(* Logix 5000 project; controller LeakTestAuto vendor 1 type 14 code 226 rev 37.11; software revision 37.01; part 13 of 15 *)
(* tags used below, declared in another part *)
   AOI_CapShuffle_Seq : AOI_Sequencer_x64;
   AOI_CTS1 : AOI_CTS_INSTRUMENT;
   AOI_CTS2 : AOI_CTS_INSTRUMENT;
   AOI_RobotPos : AOI_RobotPositions;
   AOI_SeqSteps : AOI_StandardSeqSteps;
   BarcodeInputs : udt_KeyenceScannerInputs;
   BarcodeScanner : udt_OutputStructure;
   CapShuffle_CTS1Bad : COUNTER;
   CapShuffle_CTS1Good : COUNTER;
   CapShuffle_CTS2Bad : COUNTER;
   CapShuffle_CTS2Good : COUNTER;
   CapShuffle_Seq : udt_SequenceStructure_X64;
   Conveyor : udt_OutputStructure;
   Conveyor_Seq : udt_SequenceStructure_X64;
   ConveyorHomeCounter : COUNTER;
   CTS1_Seq : udt_SequenceStructure_X64;
   CTS2_Seq : udt_SequenceStructure_X64;
   FaultsAndWarnings : STRING[96];
   LeakTester1 : udt_OutputStructure;
   LeakTester2 : udt_OutputStructure;
   Nest1Cylinder : udt_OutputStructure;
   Nest1Empty : BOOL;
   Nest1Ready : BOOL;
   Nest2Cylinder : udt_OutputStructure;
   Nest2Empty : BOOL;
   Nest2Ready : BOOL;
   OP220 : udt_Mode;
   OP220_HomingSeq : udt_SequenceStructure_X64;
   OP220_Seq : udt_SequenceStructure_X64;
   Robot : udt_OutputStructure;
   RobotGripper : udt_OutputStructure;
   RobotInputs : udt_EpsonInputs;
   ShiftTimes : SINT[24];
   TempStrBuff : STRING[10];
   test : BOOL;
   TON_CapShuffleCTS1Delay : TIMER;
   TON_CapShuffleCTS2Delay : TIMER;
   AOI_IOCounter : AOI_IOCounter;
   I_OP220_N3_CONVEYOR_CLEAT : ALIAS FOR Local:3:I.Pt13.Data;
   I_OP220_N3_CONVEYOR_LOAD : ALIAS FOR Local:3:I.Pt12.Data;
   I_OP220_N3_CONVEYOR_UNLOAD : ALIAS FOR Local:3:I.Pt14.Data;
   I_OP220_N3_DUT_PRE_NEST_0 : ALIAS FOR Local:3:I.Pt00.Data;
   I_OP220_N3_DUT_PRE_NEST_1 : ALIAS FOR Local:3:I.Pt01.Data;
   I_OP220_N3_DUT_PRE_NEST_2 : ALIAS FOR Local:3:I.Pt02.Data;
   I_OP220_N3_MAIN_AIR_OK : ALIAS FOR Local:3:I.Pt07.Data;
   I_OP220_N3_NEST1_EXTEND : ALIAS FOR Local:3:I.Pt04.Data;
   I_OP220_N3_NEST1_HOME : ALIAS FOR Local:3:I.Pt03.Data;
   I_OP220_N3_NEST2_EXTEND : ALIAS FOR Local:3:I.Pt06.Data;
   I_OP220_N3_NEST2_HOME : ALIAS FOR Local:3:I.Pt05.Data;
   I_OP220_N3_REJECT_BIN_OK : ALIAS FOR Local:3:I.Pt09.Data;
   I_OP220_N3_REJECT_CHUTE_PART : ALIAS FOR Local:3:I.Pt10.Data;
   I_OP220_N4_AC_SURGE_OK : ALIAS FOR Local:4:I.Pt00.Data;
   I_OP220_N4_CONVEYOR_ALARM_OK : ALIAS FOR Local:4:I.Pt03.Data;
   I_OP220_N4_CONVEYOR_SPEED : ALIAS FOR Local:4:I.Pt02.Data;
   I_OP220_N4_DC_OK : ALIAS FOR Local:4:I.Pt01.Data;
   I_OP220_N4_DC_OK_PS2 : ALIAS FOR Local:4:I.Pt04.Data;
   IOCounterHasRef : BOOL;
   IOCounterLastData : INT[8];
   IOLabels : STRING[128];
   IOResetArray : INT[8];
   IOTriggerCounts : UDINT[128];
   NoData : AB:5000_DI16:I:0;
   O_OP220_N5_CONV_FWD : ALIAS FOR Local:5:O.Pt12.Data;
   O_OP220_N5_CONV_REV : ALIAS FOR Local:5:O.Pt11.Data;
   O_OP220_N5_EN_CONV_ALM_RST : ALIAS FOR Local:5:O.Pt10.Data;
   O_OP220_N5_EN_GRIPPER_GRIP : ALIAS FOR Local:5:O.Pt14.Data;
   O_OP220_N5_EN_GRIPPER_UNGRIP : ALIAS FOR Local:5:O.Pt15.Data;
   O_OP220_N5_EN_LT_BU : ALIAS FOR Local:5:O.Pt03.Data;
   O_OP220_N5_EN_LT_GN : ALIAS FOR Local:5:O.Pt00.Data;
   O_OP220_N5_EN_LT_RD : ALIAS FOR Local:5:O.Pt02.Data;
   O_OP220_N5_EN_LT_YE : ALIAS FOR Local:5:O.Pt01.Data;
   O_OP220_N5_EN_MAIN_AIR : ALIAS FOR Local:5:O.Pt04.Data;
   O_OP220_N5_EN_NEST1_EXT : ALIAS FOR Local:5:O.Pt05.Data;
   O_OP220_N5_EN_NEST1_HOME : ALIAS FOR Local:5:O.Pt06.Data;
   O_OP220_N5_EN_NEST2_EXT : ALIAS FOR Local:5:O.Pt07.Data;
   O_OP220_N5_EN_NEST2_HOME : ALIAS FOR Local:5:O.Pt08.Data;
   O_OP220_N5_EN_ROBOT_LATCHOFF : ALIAS FOR Local:5:O.Pt09.Data;
   PLC : AOI_PLC;
   SI_OP220_N1_CTRL_VLAVE_NC1 : ALIAS FOR Local:1:I.Pt04.Data;
   SI_OP220_N1_LASER_AREA_NC12 : ALIAS FOR Local:1:I.Pt00.Data;
   SI_OP220_N1_LASER_GUARD_NC12 : ALIAS FOR Local:1:I.Pt01.Data;
   SI_OP220_N1_SSR_12 : ALIAS FOR Local:1:I.Pt03.Data;
   SO_OP220_N2_SSR_1 : ALIAS FOR Local:2:O.Pt00.Data;
   SO_OP220_N2_SSR_2 : ALIAS FOR Local:2:O.Pt01.Data;
(* MainProgram, continued *)

ROUTINE R98_IOCounter   (* ladder *)
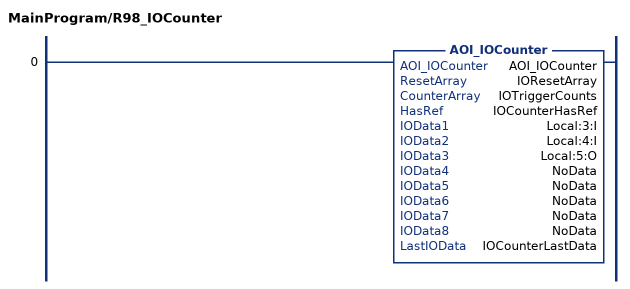
   0: AOI_IOCounter(AOI_IOCounter,IOResetArray,IOTriggerCounts,IOCounterHasRef,Local:3:I,Local:4:I,Local:5:O,NoData,NoData,NoData,NoData,NoData,IOCounterLastData);
END_ROUTINE

ROUTINE R999_SetConstants   (* structured text *)
   if PLC.FirstScan then
   	// [1] IB8S
   	IOLabels[000] := 'SI_OP220_N1_LASER_AREA_NC12';
   	IOLabels[001] := 'SI_OP220_N1_LASER_GUARD_NC12';
   	IOLabels[002] := '';
   	IOLabels[003] := 'SI_OP220_N1_SSR_12';
   	IOLabels[004] := 'SI_OP220_N1_CTRL_VLAVE_NC1';
   	IOLabels[005] := '';
   	IOLabels[006] := '';
   	IOLabels[007] := '';
   	// [2] OBV8S
   	IOLabels[008] := 'SO_OP220_N2_SSR_1';
   	IOLabels[009] := 'SO_OP220_N2_SSR_2';
   	IOLabels[010] := '';
   	IOLabels[011] := '';
   	IOLabels[012] := '';
   	IOLabels[013] := '';
   	IOLabels[014] := '';
   	IOLabels[015] := '';
   	// [3] IB16
   	IOLabels[016] := 'I_OP220_N3_DUT_PRE_NEST_0';
   	IOLabels[017] := 'I_OP220_N3_DUT_PRE_NEST_1';
   	IOLabels[018] := 'I_OP220_N3_DUT_PRE_NEST_2';
   	IOLabels[019] := 'I_OP220_N3_NEST1_HOME';
   	IOLabels[020] := 'I_OP220_N3_NEST1_EXTEND';
   	IOLabels[021] := 'I_OP220_N3_NEST2_HOME';
   	IOLabels[022] := 'I_OP220_N3_NEST2_EXTEND';
   	IOLabels[023] := 'I_OP220_N3_MAIN_AIR_OK';
   	IOLabels[024] := '';
   	IOLabels[025] := 'I_OP220_N3_REJECT_BIN_OK';
   	IOLabels[026] := 'I_OP220_N3_REJECT_CHUTE_PART';
   	IOLabels[027] := '';
   	IOLabels[028] := 'I_OP220_N3_CONVEYOR_LOAD';
   	IOLabels[029] := 'I_OP220_N3_CONVEYOR_CLEAT';
   	IOLabels[030] := 'I_OP220_N3_CONVEYOR_UNLOAD';
   	IOLabels[031] := '';
   	// [4] IB16
   	IOLabels[032] := 'I_OP220_N4_AC_SURGE_OK';
   	IOLabels[033] := 'I_OP220_N4_DC_OK';
   	IOLabels[034] := 'I_OP220_N4_CONVEYOR_SPEED';
   	IOLabels[035] := 'I_OP220_N4_CONVEYOR_ALARM_OK';
   	IOLabels[036] := 'I_OP220_N4_DC_OK_PS2';
   	IOLabels[037] := '';
   	IOLabels[038] := '';
   	IOLabels[039] := '';
   	IOLabels[040] := '';
   	IOLabels[041] := '';
   	IOLabels[042] := '';
   	IOLabels[043] := '';
   	IOLabels[044] := '';
   	IOLabels[045] := '';
   	IOLabels[046] := '';
   	IOLabels[047] := '';
   	// [5] OB16
   	IOLabels[048] := 'O_OP220_N5_EN_LT_GN';
   	IOLabels[049] := 'O_OP220_N5_EN_LT_YE';
   	IOLabels[050] := 'O_OP220_N5_EN_LT_RD';
   	IOLabels[051] := 'O_OP220_N5_EN_LT_BU';
   	IOLabels[052] := 'O_OP220_N5_EN_MAIN_AIR';
   	IOLabels[053] := 'O_OP220_N5_EN_NEST1_EXT';
   	IOLabels[054] := 'O_OP220_N5_EN_NEST1_HOME';
   	IOLabels[055] := 'O_OP220_N5_EN_NEST2_EXT';
   	IOLabels[056] := 'O_OP220_N5_EN_NEST2_HOME';
   	IOLabels[057] := 'O_OP220_N5_EN_ROBOT_LATCHOFF';
   	IOLabels[058] := 'O_OP220_N5_EN_CONV_ALM_RST';
   	IOLabels[059] := 'O_OP220_N5_CONV_REV';
   	IOLabels[060] := 'O_OP220_N5_CONV_FWD';
   	IOLabels[061] := '';
   	IOLabels[062] := 'O_OP220_N5_EN_GRIPPER_GRIP';
   	IOLabels[063] := 'O_OP220_N5_EN_GRIPPER_UNGRIP';
   	IOLabels[064] := '';
   	IOLabels[065] := '';
   	IOLabels[066] := '';
   	IOLabels[067] := '';
   	IOLabels[068] := '';
   	IOLabels[069] := '';
   	IOLabels[070] := '';
   	IOLabels[071] := '';
   	IOLabels[072] := '';
   	IOLabels[073] := '';
   	IOLabels[074] := '';
   	IOLabels[075] := '';
   	IOLabels[076] := '';
   	IOLabels[077] := '';
   	IOLabels[078] := '';
   	IOLabels[079] := '';
   	IOLabels[080] := '';
   	IOLabels[081] := '';
   	IOLabels[082] := '';
   	IOLabels[083] := '';
   	IOLabels[084] := '';
   	IOLabels[085] := '';
   	IOLabels[086] := '';
   	IOLabels[087] := '';
   	IOLabels[088] := '';
   	IOLabels[089] := '';
   	IOLabels[090] := '';
   	IOLabels[091] := '';
   	IOLabels[092] := '';
   	IOLabels[093] := '';
   	IOLabels[094] := '';
   	IOLabels[095] := '';
   	IOLabels[096] := '';
   	IOLabels[097] := '';
   	IOLabels[098] := '';
   	IOLabels[099] := '';
   	IOLabels[100] := '';
   	IOLabels[101] := '';
   	IOLabels[102] := '';
   	IOLabels[103] := '';
   	IOLabels[104] := '';
   	IOLabels[105] := '';
   	IOLabels[106] := '';
   	IOLabels[107] := '';
   	IOLabels[108] := '';
   	IOLabels[109] := '';
   	IOLabels[110] := '';
   	IOLabels[111] := '';
   	IOLabels[112] := '';
   	IOLabels[113] := '';
   	IOLabels[114] := '';
   	IOLabels[115] := '';
   	IOLabels[116] := '';
   	IOLabels[117] := '';
   	IOLabels[118] := '';
   	IOLabels[119] := '';
   	IOLabels[120] := '';
   	IOLabels[121] := '';
   	IOLabels[122] := '';
   	IOLabels[123] := '';
   	IOLabels[124] := '';
   	IOLabels[125] := '';
   	IOLabels[126] := '';
   	IOLabels[127] := '';
   
   	ShiftTimes[0] := 7;
   	ShiftTimes[1] := 15;
   	ShiftTimes[2] := 23;
   	ShiftTimes[3] := -1;
   	ShiftTimes[4] := -1;
   	ShiftTimes[5] := -1;
   	ShiftTimes[6] := -1;
   	ShiftTimes[7] := -1;
   	ShiftTimes[8] := -1;
   	ShiftTimes[9] := -1;
   	ShiftTimes[10] := -1;
   	ShiftTimes[11] := -1;
   	ShiftTimes[12] := -1;
   	ShiftTimes[13] := -1;
   	ShiftTimes[14] := -1;
   	ShiftTimes[15] := -1;
   	ShiftTimes[16] := -1;
   	ShiftTimes[17] := -1;
   	ShiftTimes[18] := -1;
   	ShiftTimes[19] := -1;
   	ShiftTimes[20] := -1;
   	ShiftTimes[21] := -1;
   	ShiftTimes[22] := -1;
   	ShiftTimes[23] := -1;
   
   	// System Faults
   	FaultsAndWarnings[000] := 'Main power off';
   	FaultsAndWarnings[001] := 'Main air not OK';
   	FaultsAndWarnings[002] := 'EStop high';
   	FaultsAndWarnings[003] := 'Guard doors open';
   	FaultsAndWarnings[004] := 'Reject bin missing';
   	FaultsAndWarnings[005] := 'No EIP connection to barcode scanner';
   	FaultsAndWarnings[006] := 'No EIP connection to CTS1';
   	FaultsAndWarnings[007] := 'No EIP connection to CTS2';
   	FaultsAndWarnings[008] := 'No EIP connection to Robot';
   	FaultsAndWarnings[009] := 'EStop Safety Block faulted';
   	FaultsAndWarnings[010] := 'Barcode scanner fault';
   	FaultsAndWarnings[011] := 'CTS1 fault';
   	FaultsAndWarnings[012] := 'CTS2 fault';
   	FaultsAndWarnings[013] := 'Robot fault';
   	FaultsAndWarnings[014] := 'Robot gripper in unknown state';
   	FaultsAndWarnings[015] := 'Conveyor alarm high';
   	FaultsAndWarnings[016] := 'Cylinder 1 fault';
   	FaultsAndWarnings[017] := 'Cylinder 2 fault';
   	FaultsAndWarnings[018] := '24V DC not OK';
   	FaultsAndWarnings[019] := 'Check conveyor cleat sensor';
   	FaultsAndWarnings[020] := '';
   	FaultsAndWarnings[021] := '';
   	FaultsAndWarnings[022] := '';
   	FaultsAndWarnings[023] := '';
   	FaultsAndWarnings[024] := '';
   	FaultsAndWarnings[025] := '';
   	FaultsAndWarnings[026] := '';
   	FaultsAndWarnings[027] := '';
   	FaultsAndWarnings[028] := '';
   	FaultsAndWarnings[029] := '';
   	FaultsAndWarnings[030] := '';
   	FaultsAndWarnings[031] := '';
   	// Sequence Faults
   	FaultsAndWarnings[032] := '3 in a row fault';
   	FaultsAndWarnings[033] := '5 in an hour fault';
   	FaultsAndWarnings[034] := '10 in a shift fault';
   	FaultsAndWarnings[035] := '';
   	FaultsAndWarnings[036] := '';
   	FaultsAndWarnings[037] := '';
   	FaultsAndWarnings[038] := '';
   	FaultsAndWarnings[039] := '';
   	FaultsAndWarnings[040] := '';
   	FaultsAndWarnings[041] := '';
   	FaultsAndWarnings[042] := 'Homing cycle overtime';
   	FaultsAndWarnings[043] := 'Fail chute failed to register unit (Homing Seq)';
   	FaultsAndWarnings[044] := 'Fail chute failed to register unit (Auto Seq)';
   	FaultsAndWarnings[045] := 'Cylinder 1 down timeout';
   	FaultsAndWarnings[046] := 'Cylinder 2 down timeout';
   	FaultsAndWarnings[047] := 'Cylinder 1 up timeout';
   	FaultsAndWarnings[048] := 'Cylinder 2 up timeout';
   	FaultsAndWarnings[049] := 'Cylinder 1 movement requested but RFID not matching expected value.';
   	FaultsAndWarnings[050] := 'Cylinder 2 movement requested but RFID not matching expected value.';
   	FaultsAndWarnings[051] := '';
   	FaultsAndWarnings[052] := '';
   	FaultsAndWarnings[053] := '';
   	FaultsAndWarnings[054] := '';
   	FaultsAndWarnings[055] := '';
   	FaultsAndWarnings[056] := '';
   	FaultsAndWarnings[057] := '';
   	FaultsAndWarnings[058] := '';
   	FaultsAndWarnings[059] := '';
   	FaultsAndWarnings[060] := '';
   	FaultsAndWarnings[061] := '';
   	FaultsAndWarnings[062] := '';
   	FaultsAndWarnings[063] := '';
   	// Warnings
   	FaultsAndWarnings[064] := 'Cycle stop requested';
   	FaultsAndWarnings[065] := 'Cycle pause requested';
   	FaultsAndWarnings[066] := 'Step mode active';
   	FaultsAndWarnings[067] := 'Dry cycle active';
   	FaultsAndWarnings[068] := 'MES bypass active';
   	FaultsAndWarnings[069] := '';
   	FaultsAndWarnings[070] := '';
   	FaultsAndWarnings[071] := '';
   	FaultsAndWarnings[072] := '';
   	FaultsAndWarnings[073] := '';
   	FaultsAndWarnings[074] := 'Main sequence stuck on step$n';
   	FaultsAndWarnings[075] := 'Homing sequence stuck on step$n';
   	FaultsAndWarnings[076] := 'CTS1 sequence stuck on step ';
   	FaultsAndWarnings[077] := 'CTS2 sequence stuck on step ';
   	FaultsAndWarnings[078] := 'Conveyor sequence stuck on step ';
   	FaultsAndWarnings[079] := 'Main sequence stuck on step$n';
   	FaultsAndWarnings[080] := 'Homing sequence stuck on step$n';
   	FaultsAndWarnings[081] := 'CTS1 sequence stuck on step ';
   	FaultsAndWarnings[082] := 'CTS2 sequence stuck on step ';
   	FaultsAndWarnings[083] := 'Conveyor sequence stuck on step ';
   	FaultsAndWarnings[084] := 'CTS1 test requested but interlock not met';
   	FaultsAndWarnings[085] := 'CTS2 test requested but interlock not met';
   	FaultsAndWarnings[086] := 'CTS1 not ready';
   	FaultsAndWarnings[087] := 'CTS2 not ready';
   	FaultsAndWarnings[088] := 'Robot movement requested but interlock not met';
   	FaultsAndWarnings[089] := 'Conveyor movement requested but interlock not met';
   	FaultsAndWarnings[090] := 'Nest 1 movement requested but interlock not met';
   	FaultsAndWarnings[091] := 'Nest 2 movement requested but interlock not met';
   	FaultsAndWarnings[092] := '';
   	FaultsAndWarnings[093] := '';
   	FaultsAndWarnings[094] := 'Fail bin full, please empty';
   	FaultsAndWarnings[095] := '';
   end_if;
   
   // Done this way because concat cannot accept string literals
   // DTOS(OP220_Seq.CurrentStep,TempStrBuff[0]);
   // CONCAT(FaultsAndWarnings[079], TempStrBuff[0], FaultsAndWarnings[074]);
   CONCAT(FaultsAndWarnings[079], OP220_Seq.HMI_CurrentStepDescription, FaultsAndWarnings[074]);
   // DTOS(OP220_HomingSeq.CurrentStep,TempStrBuff[0]);
   // CONCAT(FaultsAndWarnings[080], TempStrBuff[0], FaultsAndWarnings[075]);
   CONCAT(FaultsAndWarnings[080], OP220_HomingSeq.HMI_CurrentStepDescription, FaultsAndWarnings[075]);
   DTOS(CTS1_Seq.CurrentStep,TempStrBuff[0]);
   CONCAT(FaultsAndWarnings[081], TempStrBuff[0], FaultsAndWarnings[076]);
   DTOS(CTS2_Seq.CurrentStep,TempStrBuff[0]);
   CONCAT(FaultsAndWarnings[082], TempStrBuff[0], FaultsAndWarnings[077]);
   DTOS(Conveyor_Seq.CurrentStep,TempStrBuff[0]);
   CONCAT(FaultsAndWarnings[083], TempStrBuff[0], FaultsAndWarnings[078]);
   
   AOI_RobotPositions(AOI_RobotPos);
   AOI_StandardSeqSteps(AOI_SeqSteps);
END_ROUTINE

ROUTINE R99_StepDescriptions   (* structured text *)
   case OP220_Seq.CurrentStep of
   	1000:
   		OP220_Seq.HMI_CurrentStepDescription := 'Waiting for next action';
   	2000,2010,2500,2510:
   		OP220_Seq.HMI_CurrentStepDescription := 'Pick up DUT from load nest';
   	2020,2030,2520,2530:
   		OP220_Seq.HMI_CurrentStepDescription := 'Scan DUT barcode';
   	2040,2050,2060:
   		OP220_Seq.HMI_CurrentStepDescription := 'Load DUT to nest 1';
   	2540,2550,2560:
   		OP220_Seq.HMI_CurrentStepDescription := 'Load DUT to nest 2';
   	2070,2080:
   		OP220_Seq.HMI_CurrentStepDescription := 'Start leak test nest 1';
   	2570,2580:
   		OP220_Seq.HMI_CurrentStepDescription := 'Start leak test nest 2';
   	3000,3010:
   		OP220_Seq.HMI_CurrentStepDescription := 'Pick up DUT from nest 1';
   	3500,3510:
   		OP220_Seq.HMI_CurrentStepDescription := 'Pick up DUT from nest 2';
   	3020,3520:
   		OP220_Seq.HMI_CurrentStepDescription := 'Drop off DUT';
   	3030,3040,3530,3540:
   		OP220_Seq.HMI_CurrentStepDescription := 'Drop off DUT at conveyor';
   	3050,3550:
   		OP220_Seq.HMI_CurrentStepDescription := 'Index conveyor';
   	7000,7010:
   		OP220_Seq.HMI_CurrentStepDescription := 'Drop off DUT at fail chute (Barcode)';
   	7100,7110:
   		OP220_Seq.HMI_CurrentStepDescription := 'Drop off DUT at fail chute (Nest 1)';
   	7200,7210:
   		OP220_Seq.HMI_CurrentStepDescription := 'Drop off DUT at fail chute (Nest 2)';
   	else
   		OP220_Seq.HMI_CurrentStepDescription := '';
   end_case;
   
   case OP220_HomingSeq.CurrentStep of
   	1000,1010:
   		OP220_HomingSeq.HMI_CurrentStepDescription := 'Drop gripped DUT to fail chute';
   	1020,1030:
   		OP220_HomingSeq.HMI_CurrentStepDescription := 'Move nest cylinders to home position';
   	1040,1050,1060,1070:
   		OP220_HomingSeq.HMI_CurrentStepDescription := 'Unload nest 1 to fail chute';
   	1080,1090,1100,1110:
   		OP220_HomingSeq.HMI_CurrentStepDescription := 'Unload nest 2 to fail chute';
   	1120,1130:
   		OP220_HomingSeq.HMI_CurrentStepDescription := 'Move robot to scanner';
   	1140,1150:
   		OP220_HomingSeq.HMI_CurrentStepDescription := 'Check conveyor empty (';
   		DTOS(ConveyorHomeCounter.ACC, TempStrBuff[0]);
   		TempStrBuff[1] := '/';
   		DTOS(ConveyorHomeCounter.PRE, TempStrBuff[2]);
   		TempStrBuff[3] := ')';
   		CONCAT(OP220_HomingSeq.HMI_CurrentStepDescription, TempStrBuff[0], OP220_HomingSeq.HMI_CurrentStepDescription);
   		CONCAT(OP220_HomingSeq.HMI_CurrentStepDescription, TempStrBuff[1], OP220_HomingSeq.HMI_CurrentStepDescription);
   		CONCAT(OP220_HomingSeq.HMI_CurrentStepDescription, TempStrBuff[2], OP220_HomingSeq.HMI_CurrentStepDescription);
   		CONCAT(OP220_HomingSeq.HMI_CurrentStepDescription, TempStrBuff[3], OP220_HomingSeq.HMI_CurrentStepDescription);
   	else
   		OP220_HomingSeq.HMI_CurrentStepDescription := '';
   end_case;
END_ROUTINE

ROUTINE zR10_CapShuffle   (* ladder *)
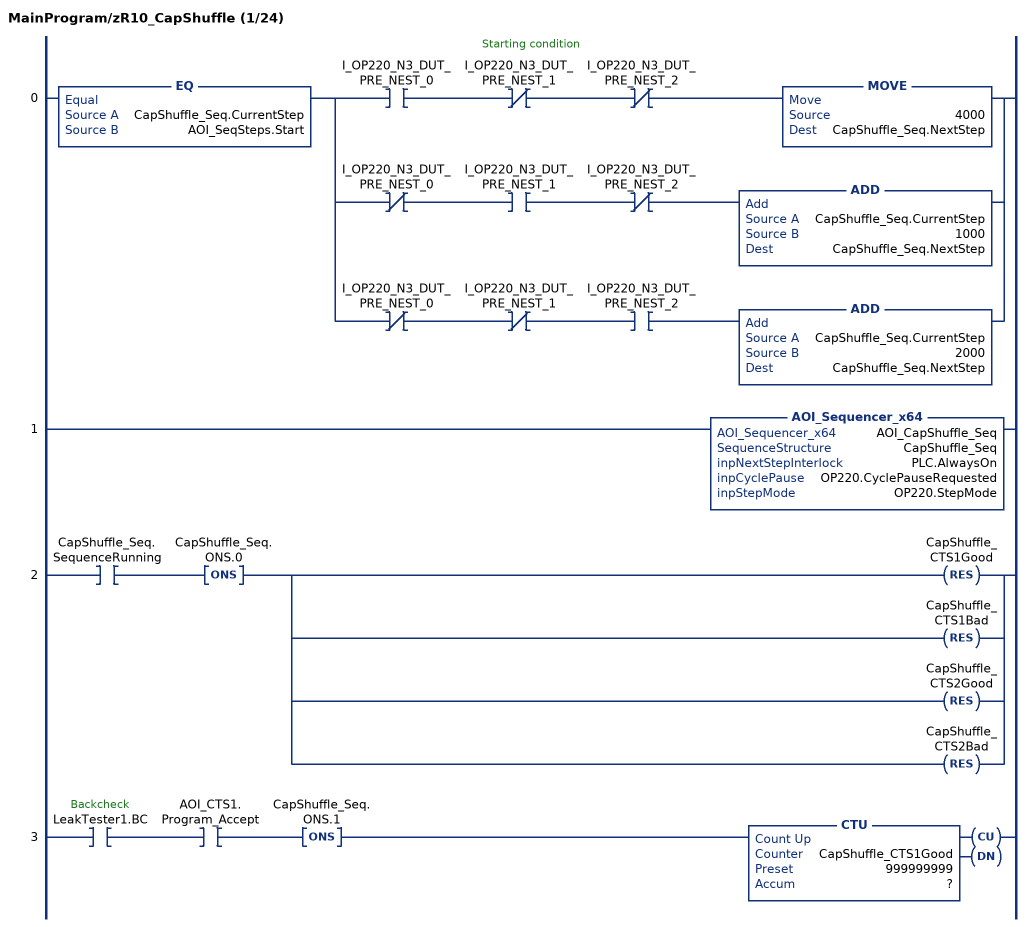
   // Starting condition
   0: EQ(CapShuffle_Seq.CurrentStep,AOI_SeqSteps.Start)[XIC(I_OP220_N3_DUT_PRE_NEST_0) XIO(I_OP220_N3_DUT_PRE_NEST_1) XIO(I_OP220_N3_DUT_PRE_NEST_2) MOVE(4000,CapShuffle_Seq.NextStep) ,XIO(I_OP220_N3_DUT_PRE_NEST_0) XIC(I_OP220_N3_DUT_PRE_NEST_1) XIO(I_OP220_N3_DUT_PRE_NEST_2) ADD(CapShuffle_Seq.CurrentStep,1000,CapShuffle_Seq.NextStep) ,XIO(I_OP220_N3_DUT_PRE_NEST_0) XIO(I_OP220_N3_DUT_PRE_NEST_1) XIC(I_OP220_N3_DUT_PRE_NEST_2) ADD(CapShuffle_Seq.CurrentStep,2000,CapShuffle_Seq.NextStep) ];
   1: AOI_Sequencer_x64(AOI_CapShuffle_Seq,CapShuffle_Seq,PLC.AlwaysOn,OP220.CyclePauseRequested,OP220.StepMode);
   2: XIC(CapShuffle_Seq.SequenceRunning)ONS(CapShuffle_Seq.ONS.0)[RES(CapShuffle_CTS1Good) ,RES(CapShuffle_CTS1Bad) ,RES(CapShuffle_CTS2Good) ,RES(CapShuffle_CTS2Bad) ];
   3: XIC(LeakTester1.BC)XIC(AOI_CTS1.Program_Accept)ONS(CapShuffle_Seq.ONS.1)CTU(CapShuffle_CTS1Good,?,?);
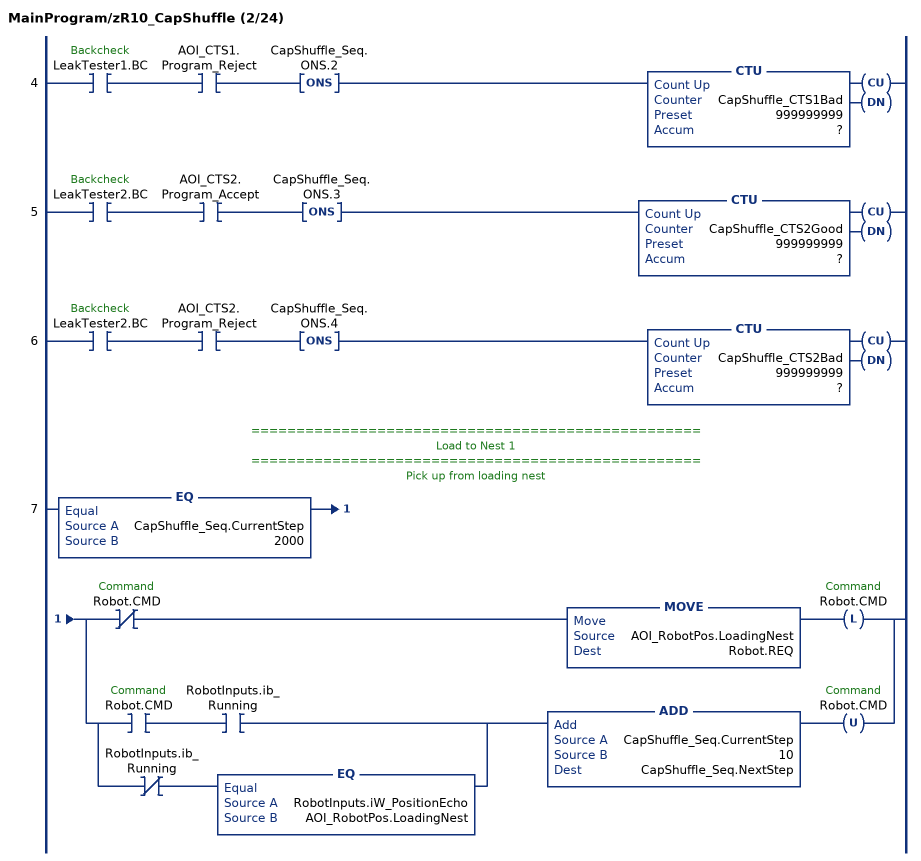
   4: XIC(LeakTester1.BC)XIC(AOI_CTS1.Program_Reject)ONS(CapShuffle_Seq.ONS.2)CTU(CapShuffle_CTS1Bad,?,?);
   5: XIC(LeakTester2.BC)XIC(AOI_CTS2.Program_Accept)ONS(CapShuffle_Seq.ONS.3)CTU(CapShuffle_CTS2Good,?,?);
   6: XIC(LeakTester2.BC)XIC(AOI_CTS2.Program_Reject)ONS(CapShuffle_Seq.ONS.4)CTU(CapShuffle_CTS2Bad,?,?);
   // ==================================================
   // Load to Nest 1
   // ==================================================
   // Pick up from loading nest
   7: EQ(CapShuffle_Seq.CurrentStep,2000)[XIO(Robot.CMD) MOVE(AOI_RobotPos.LoadingNest,Robot.REQ) OTL(Robot.CMD) ,[XIC(Robot.CMD) XIC(RobotInputs.ib_Running) ,XIO(RobotInputs.ib_Running) EQ(RobotInputs.iW_PositionEcho,AOI_RobotPos.LoadingNest) ] ADD(CapShuffle_Seq.CurrentStep,10,CapShuffle_Seq.NextStep) OTU(Robot.CMD) ];
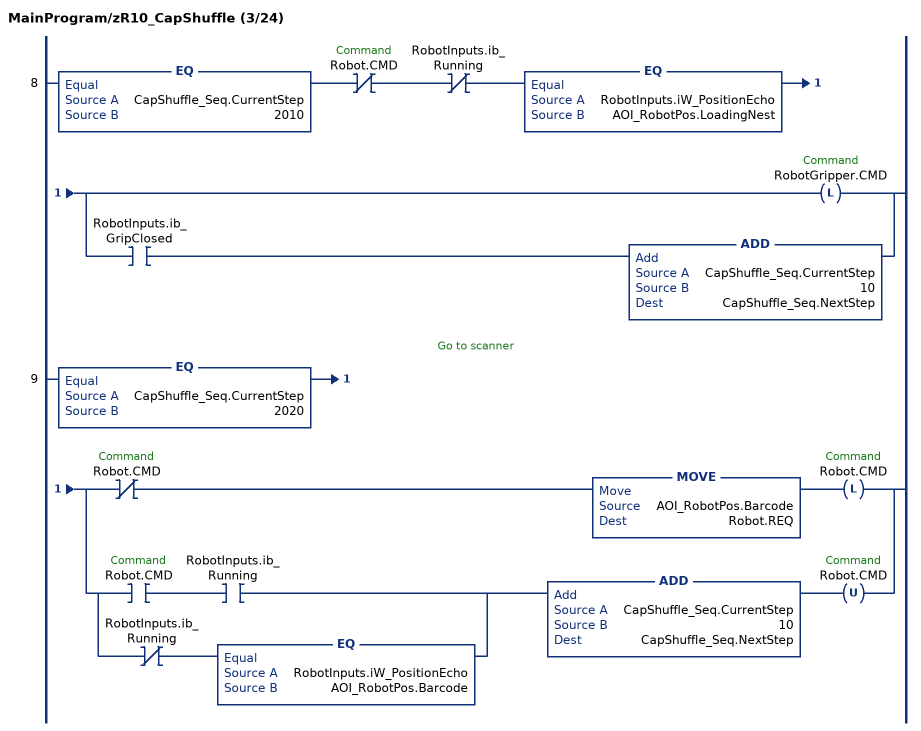
   8: EQ(CapShuffle_Seq.CurrentStep,2010)XIO(Robot.CMD)XIO(RobotInputs.ib_Running)EQ(RobotInputs.iW_PositionEcho,AOI_RobotPos.LoadingNest)[OTL(RobotGripper.CMD) ,XIC(RobotInputs.ib_GripClosed) ADD(CapShuffle_Seq.CurrentStep,10,CapShuffle_Seq.NextStep) ];
   // Go to scanner
   9: EQ(CapShuffle_Seq.CurrentStep,2020)[XIO(Robot.CMD) MOVE(AOI_RobotPos.Barcode,Robot.REQ) OTL(Robot.CMD) ,[XIC(Robot.CMD) XIC(RobotInputs.ib_Running) ,XIO(RobotInputs.ib_Running) EQ(RobotInputs.iW_PositionEcho,AOI_RobotPos.Barcode) ] ADD(CapShuffle_Seq.CurrentStep,10,CapShuffle_Seq.NextStep) OTU(Robot.CMD) ];
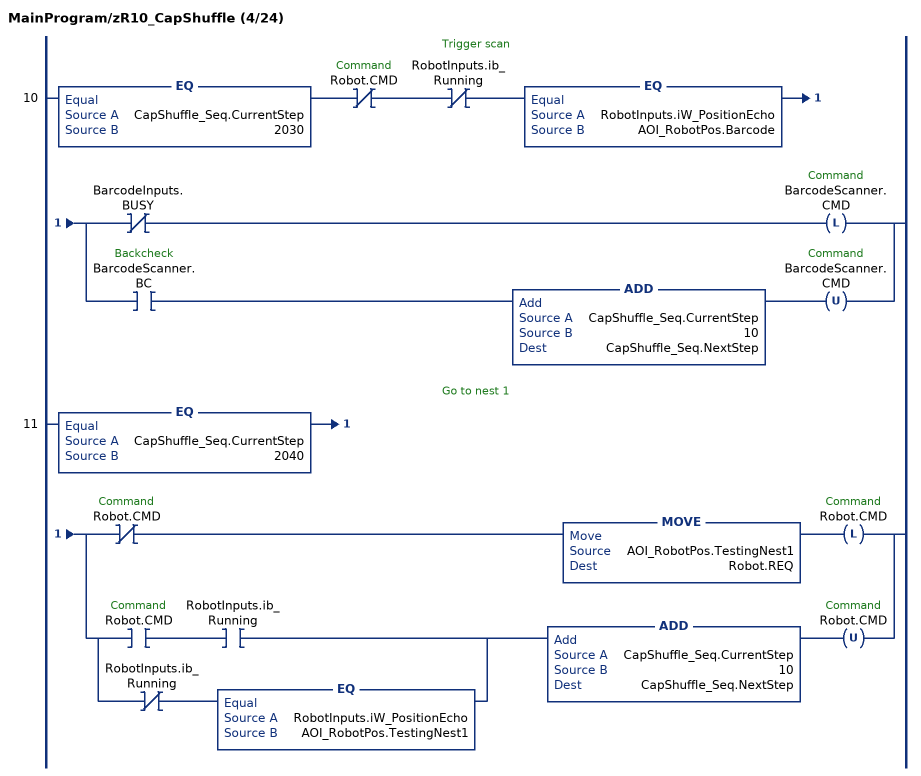
   // Trigger scan
   10: EQ(CapShuffle_Seq.CurrentStep,2030)XIO(Robot.CMD)XIO(RobotInputs.ib_Running)EQ(RobotInputs.iW_PositionEcho,AOI_RobotPos.Barcode)[XIO(BarcodeInputs.BUSY) OTL(BarcodeScanner.CMD) ,XIC(BarcodeScanner.BC) ADD(CapShuffle_Seq.CurrentStep,10,CapShuffle_Seq.NextStep) OTU(BarcodeScanner.CMD) ];
   // Go to nest 1
   11: EQ(CapShuffle_Seq.CurrentStep,2040)[XIO(Robot.CMD) MOVE(AOI_RobotPos.TestingNest1,Robot.REQ) OTL(Robot.CMD) ,[XIC(Robot.CMD) XIC(RobotInputs.ib_Running) ,XIO(RobotInputs.ib_Running) EQ(RobotInputs.iW_PositionEcho,AOI_RobotPos.TestingNest1) ] ADD(CapShuffle_Seq.CurrentStep,10,CapShuffle_Seq.NextStep) OTU(Robot.CMD) ];
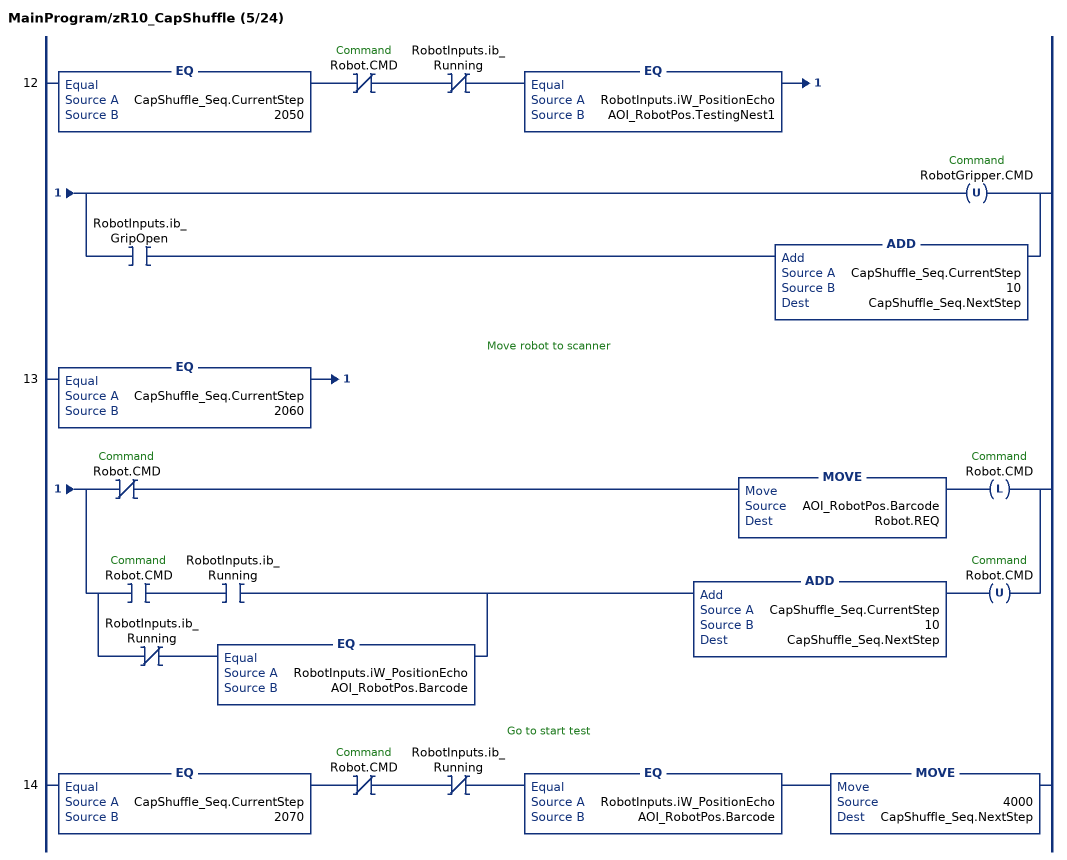
   12: EQ(CapShuffle_Seq.CurrentStep,2050)XIO(Robot.CMD)XIO(RobotInputs.ib_Running)EQ(RobotInputs.iW_PositionEcho,AOI_RobotPos.TestingNest1)[OTU(RobotGripper.CMD) ,XIC(RobotInputs.ib_GripOpen) ADD(CapShuffle_Seq.CurrentStep,10,CapShuffle_Seq.NextStep) ];
   // Move robot to scanner
   13: EQ(CapShuffle_Seq.CurrentStep,2060)[XIO(Robot.CMD) MOVE(AOI_RobotPos.Barcode,Robot.REQ) OTL(Robot.CMD) ,[XIC(Robot.CMD) XIC(RobotInputs.ib_Running) ,XIO(RobotInputs.ib_Running) EQ(RobotInputs.iW_PositionEcho,AOI_RobotPos.Barcode) ] ADD(CapShuffle_Seq.CurrentStep,10,CapShuffle_Seq.NextStep) OTU(Robot.CMD) ];
   // Go to start test
   14: EQ(CapShuffle_Seq.CurrentStep,2070)XIO(Robot.CMD)XIO(RobotInputs.ib_Running)EQ(RobotInputs.iW_PositionEcho,AOI_RobotPos.Barcode)MOVE(4000,CapShuffle_Seq.NextStep);
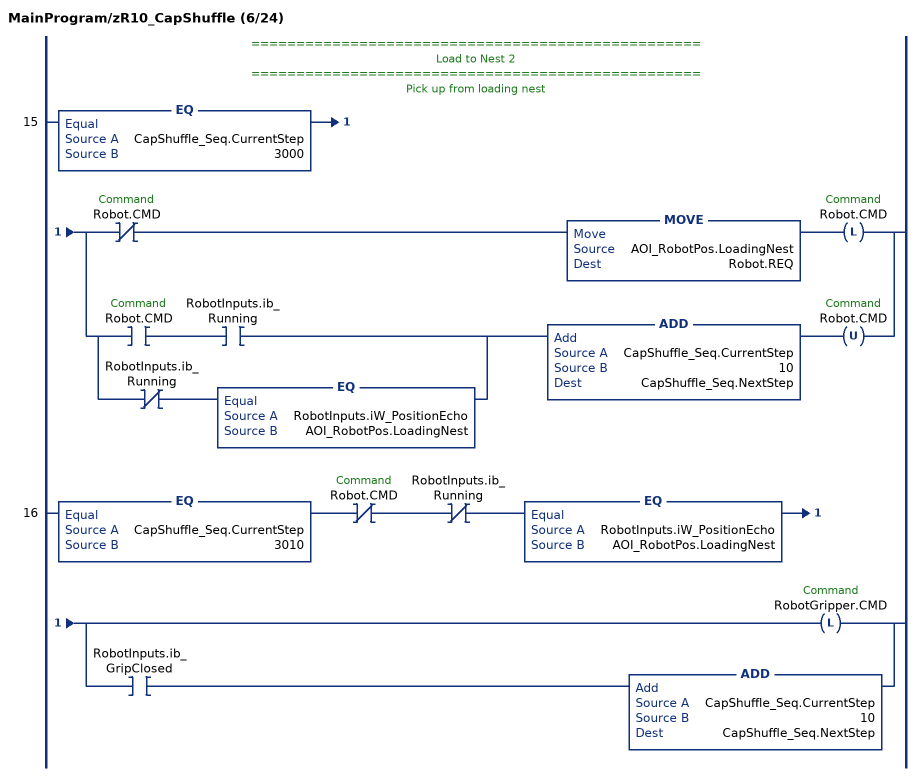
   // ==================================================
   // Load to Nest 2
   // ==================================================
   // Pick up from loading nest
   15: EQ(CapShuffle_Seq.CurrentStep,3000)[XIO(Robot.CMD) MOVE(AOI_RobotPos.LoadingNest,Robot.REQ) OTL(Robot.CMD) ,[XIC(Robot.CMD) XIC(RobotInputs.ib_Running) ,XIO(RobotInputs.ib_Running) EQ(RobotInputs.iW_PositionEcho,AOI_RobotPos.LoadingNest) ] ADD(CapShuffle_Seq.CurrentStep,10,CapShuffle_Seq.NextStep) OTU(Robot.CMD) ];
   16: EQ(CapShuffle_Seq.CurrentStep,3010)XIO(Robot.CMD)XIO(RobotInputs.ib_Running)EQ(RobotInputs.iW_PositionEcho,AOI_RobotPos.LoadingNest)[OTL(RobotGripper.CMD) ,XIC(RobotInputs.ib_GripClosed) ADD(CapShuffle_Seq.CurrentStep,10,CapShuffle_Seq.NextStep) ];
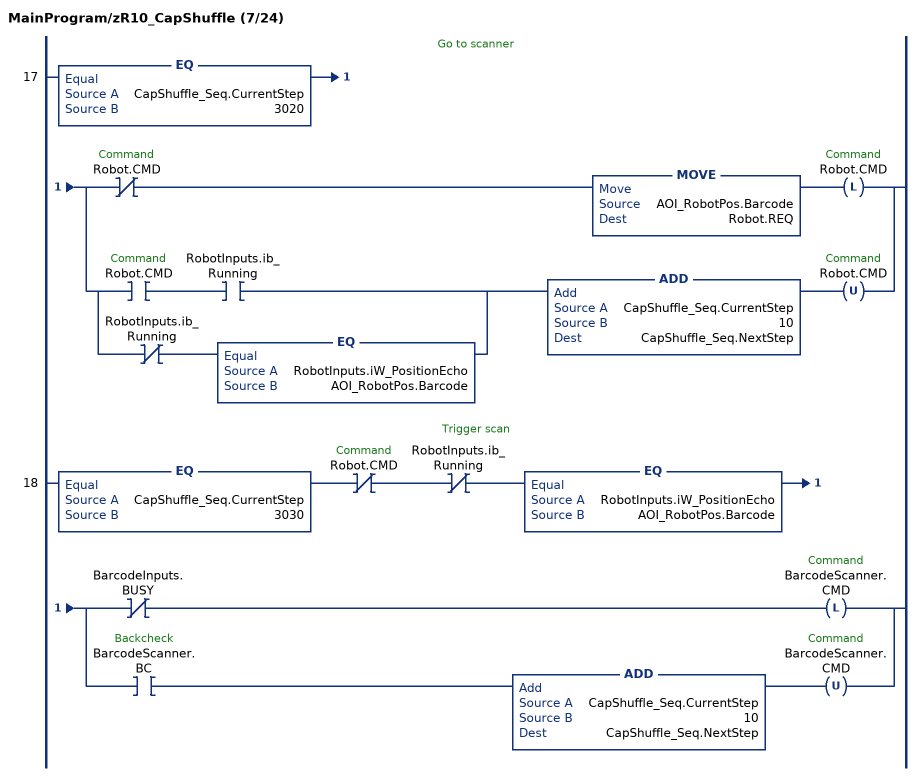
   // Go to scanner
   17: EQ(CapShuffle_Seq.CurrentStep,3020)[XIO(Robot.CMD) MOVE(AOI_RobotPos.Barcode,Robot.REQ) OTL(Robot.CMD) ,[XIC(Robot.CMD) XIC(RobotInputs.ib_Running) ,XIO(RobotInputs.ib_Running) EQ(RobotInputs.iW_PositionEcho,AOI_RobotPos.Barcode) ] ADD(CapShuffle_Seq.CurrentStep,10,CapShuffle_Seq.NextStep) OTU(Robot.CMD) ];
   // Trigger scan
   18: EQ(CapShuffle_Seq.CurrentStep,3030)XIO(Robot.CMD)XIO(RobotInputs.ib_Running)EQ(RobotInputs.iW_PositionEcho,AOI_RobotPos.Barcode)[XIO(BarcodeInputs.BUSY) OTL(BarcodeScanner.CMD) ,XIC(BarcodeScanner.BC) ADD(CapShuffle_Seq.CurrentStep,10,CapShuffle_Seq.NextStep) OTU(BarcodeScanner.CMD) ];
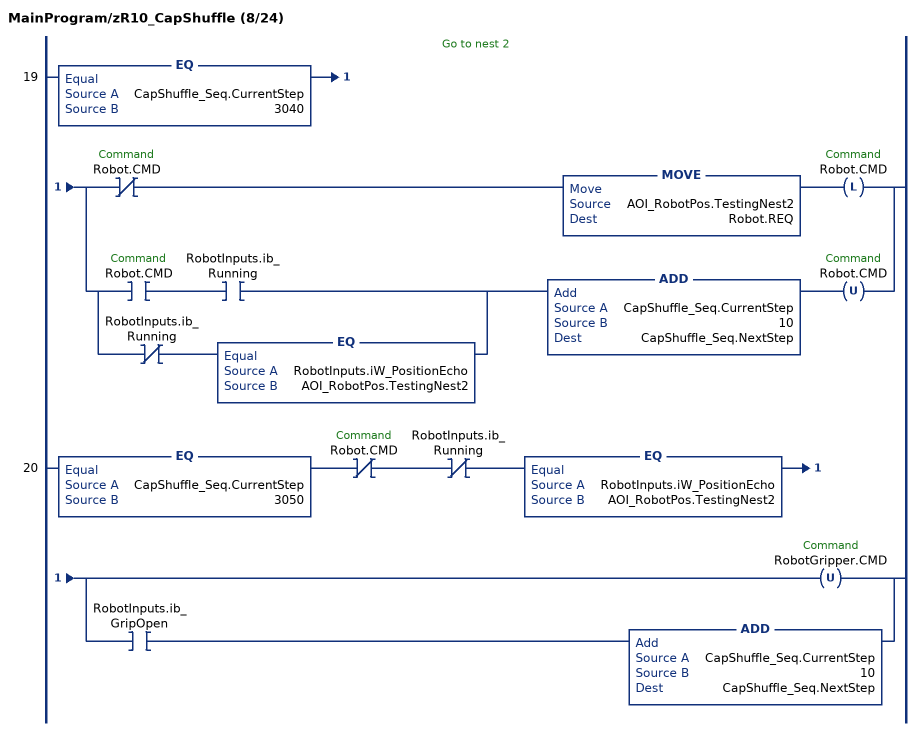
   // Go to nest 2
   19: EQ(CapShuffle_Seq.CurrentStep,3040)[XIO(Robot.CMD) MOVE(AOI_RobotPos.TestingNest2,Robot.REQ) OTL(Robot.CMD) ,[XIC(Robot.CMD) XIC(RobotInputs.ib_Running) ,XIO(RobotInputs.ib_Running) EQ(RobotInputs.iW_PositionEcho,AOI_RobotPos.TestingNest2) ] ADD(CapShuffle_Seq.CurrentStep,10,CapShuffle_Seq.NextStep) OTU(Robot.CMD) ];
   20: EQ(CapShuffle_Seq.CurrentStep,3050)XIO(Robot.CMD)XIO(RobotInputs.ib_Running)EQ(RobotInputs.iW_PositionEcho,AOI_RobotPos.TestingNest2)[OTU(RobotGripper.CMD) ,XIC(RobotInputs.ib_GripOpen) ADD(CapShuffle_Seq.CurrentStep,10,CapShuffle_Seq.NextStep) ];
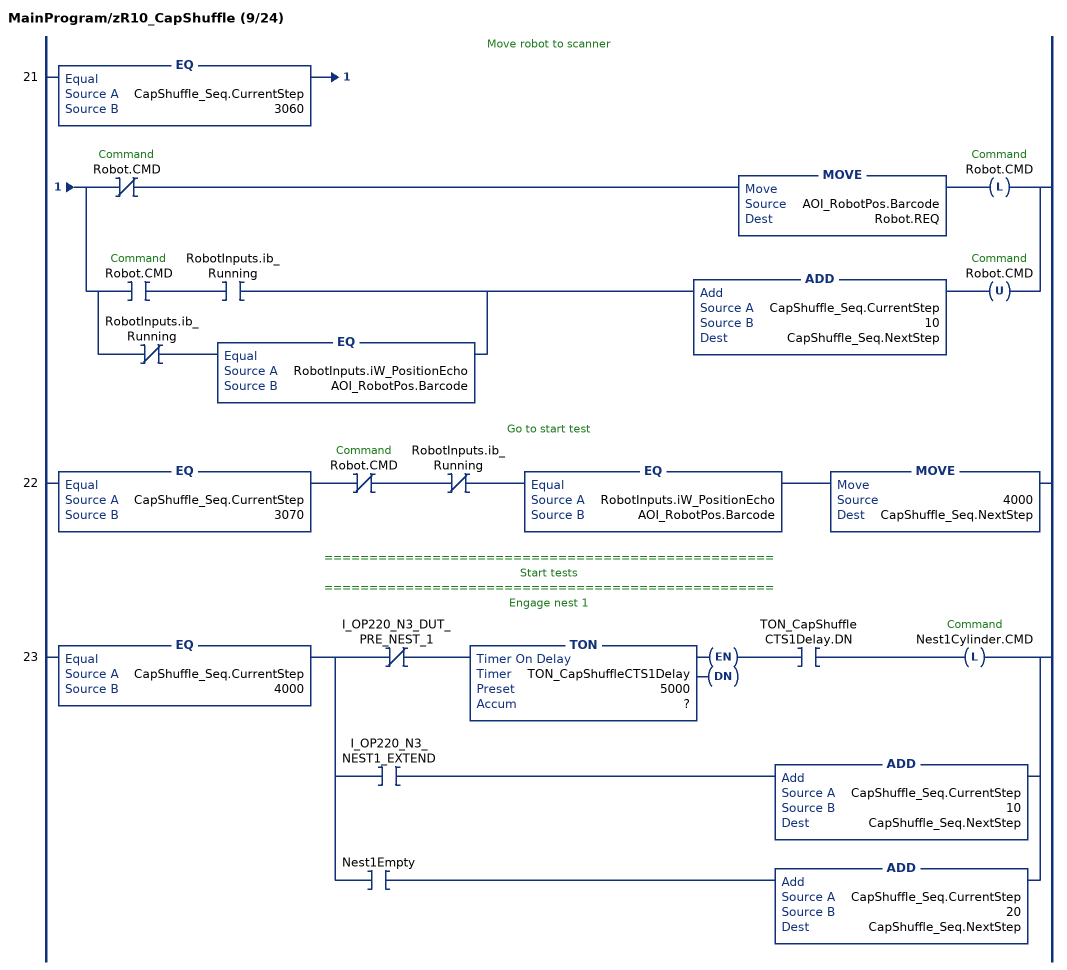
   // Move robot to scanner
   21: EQ(CapShuffle_Seq.CurrentStep,3060)[XIO(Robot.CMD) MOVE(AOI_RobotPos.Barcode,Robot.REQ) OTL(Robot.CMD) ,[XIC(Robot.CMD) XIC(RobotInputs.ib_Running) ,XIO(RobotInputs.ib_Running) EQ(RobotInputs.iW_PositionEcho,AOI_RobotPos.Barcode) ] ADD(CapShuffle_Seq.CurrentStep,10,CapShuffle_Seq.NextStep) OTU(Robot.CMD) ];
   // Go to start test
   22: EQ(CapShuffle_Seq.CurrentStep,3070)XIO(Robot.CMD)XIO(RobotInputs.ib_Running)EQ(RobotInputs.iW_PositionEcho,AOI_RobotPos.Barcode)MOVE(4000,CapShuffle_Seq.NextStep);
   // ==================================================
   // Start tests
   // ==================================================
   // Engage nest 1
   23: EQ(CapShuffle_Seq.CurrentStep,4000)[XIO(I_OP220_N3_DUT_PRE_NEST_1) TON(TON_CapShuffleCTS1Delay,?,?) XIC(TON_CapShuffleCTS1Delay.DN) OTL(Nest1Cylinder.CMD) ,XIC(I_OP220_N3_NEST1_EXTEND) ADD(CapShuffle_Seq.CurrentStep,10,CapShuffle_Seq.NextStep) ,XIC(Nest1Empty) ADD(CapShuffle_Seq.CurrentStep,20,CapShuffle_Seq.NextStep) ];
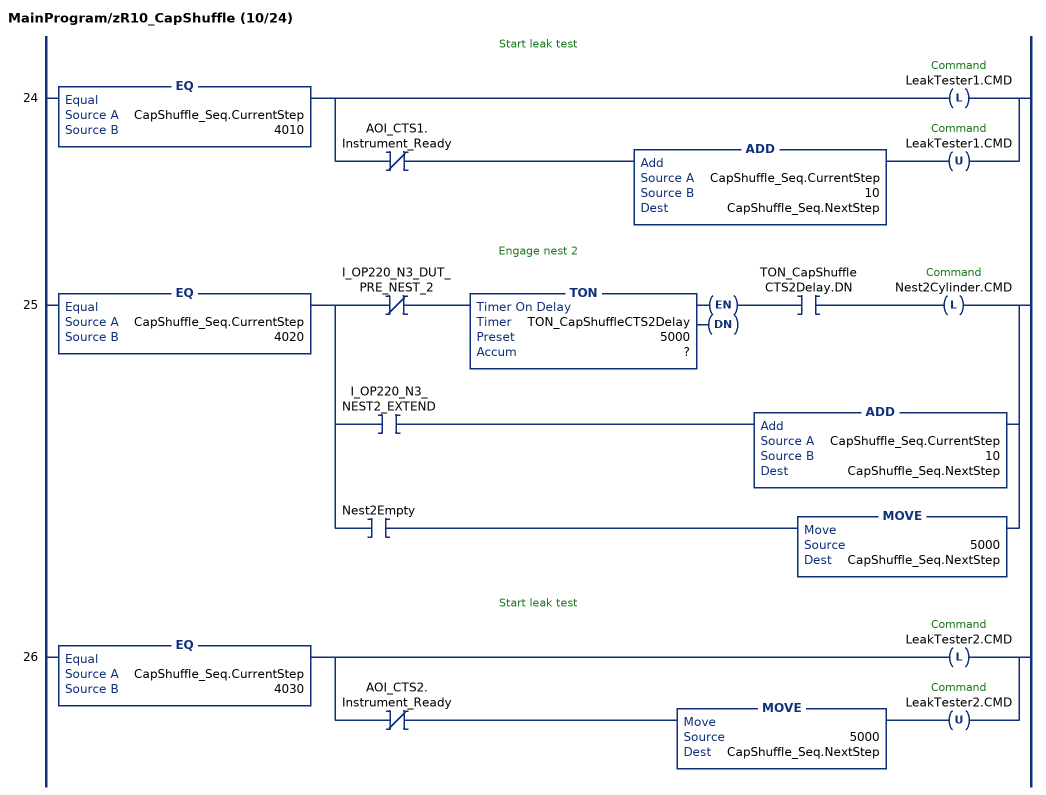
   // Start leak test
   24: EQ(CapShuffle_Seq.CurrentStep,4010)[OTL(LeakTester1.CMD) ,XIO(AOI_CTS1.Instrument_Ready) ADD(CapShuffle_Seq.CurrentStep,10,CapShuffle_Seq.NextStep) OTU(LeakTester1.CMD) ];
   // Engage nest 2
   25: EQ(CapShuffle_Seq.CurrentStep,4020)[XIO(I_OP220_N3_DUT_PRE_NEST_2) TON(TON_CapShuffleCTS2Delay,?,?) XIC(TON_CapShuffleCTS2Delay.DN) OTL(Nest2Cylinder.CMD) ,XIC(I_OP220_N3_NEST2_EXTEND) ADD(CapShuffle_Seq.CurrentStep,10,CapShuffle_Seq.NextStep) ,XIC(Nest2Empty) MOVE(5000,CapShuffle_Seq.NextStep) ];
   // Start leak test
   26: EQ(CapShuffle_Seq.CurrentStep,4030)[OTL(LeakTester2.CMD) ,XIO(AOI_CTS2.Instrument_Ready) MOVE(5000,CapShuffle_Seq.NextStep) OTU(LeakTester2.CMD) ];
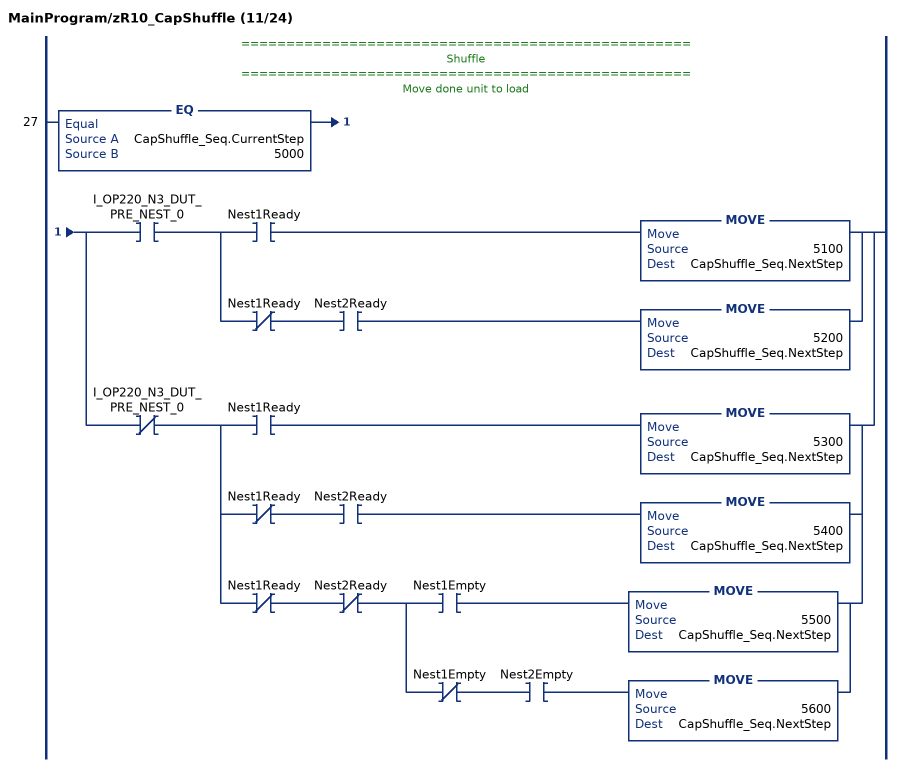
   // ==================================================
   // Shuffle
   // ==================================================
   // Move done unit to load
   27: EQ(CapShuffle_Seq.CurrentStep,5000)[XIC(I_OP220_N3_DUT_PRE_NEST_0) [XIC(Nest1Ready) MOVE(5100,CapShuffle_Seq.NextStep) ,XIO(Nest1Ready) XIC(Nest2Ready) MOVE(5200,CapShuffle_Seq.NextStep) ] ,XIO(I_OP220_N3_DUT_PRE_NEST_0) [XIC(Nest1Ready) MOVE(5300,CapShuffle_Seq.NextStep) ,XIO(Nest1Ready) XIC(Nest2Ready) MOVE(5400,CapShuffle_Seq.NextStep) ,XIO(Nest1Ready) XIO(Nest2Ready) [XIC(Nest1Empty) MOVE(5500,CapShuffle_Seq.NextStep) ,XIO(Nest1Empty) XIC(Nest2Empty) MOVE(5600,CapShuffle_Seq.NextStep) ] ] ];
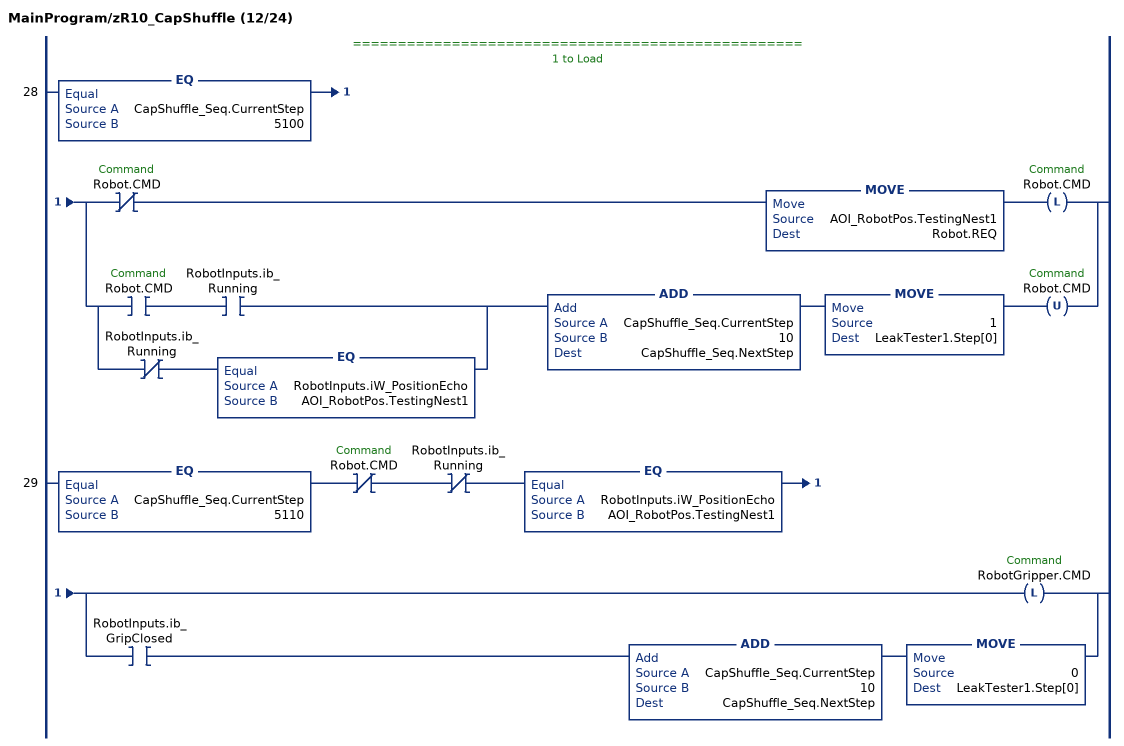
   // ==================================================
   // 1 to Load
   28: EQ(CapShuffle_Seq.CurrentStep,5100)[XIO(Robot.CMD) MOVE(AOI_RobotPos.TestingNest1,Robot.REQ) OTL(Robot.CMD) ,[XIC(Robot.CMD) XIC(RobotInputs.ib_Running) ,XIO(RobotInputs.ib_Running) EQ(RobotInputs.iW_PositionEcho,AOI_RobotPos.TestingNest1) ] ADD(CapShuffle_Seq.CurrentStep,10,CapShuffle_Seq.NextStep) MOVE(1,LeakTester1.Step[0]) OTU(Robot.CMD) ];
   29: EQ(CapShuffle_Seq.CurrentStep,5110)XIO(Robot.CMD)XIO(RobotInputs.ib_Running)EQ(RobotInputs.iW_PositionEcho,AOI_RobotPos.TestingNest1)[OTL(RobotGripper.CMD) ,XIC(RobotInputs.ib_GripClosed) ADD(CapShuffle_Seq.CurrentStep,10,CapShuffle_Seq.NextStep) MOVE(0,LeakTester1.Step[0]) ];
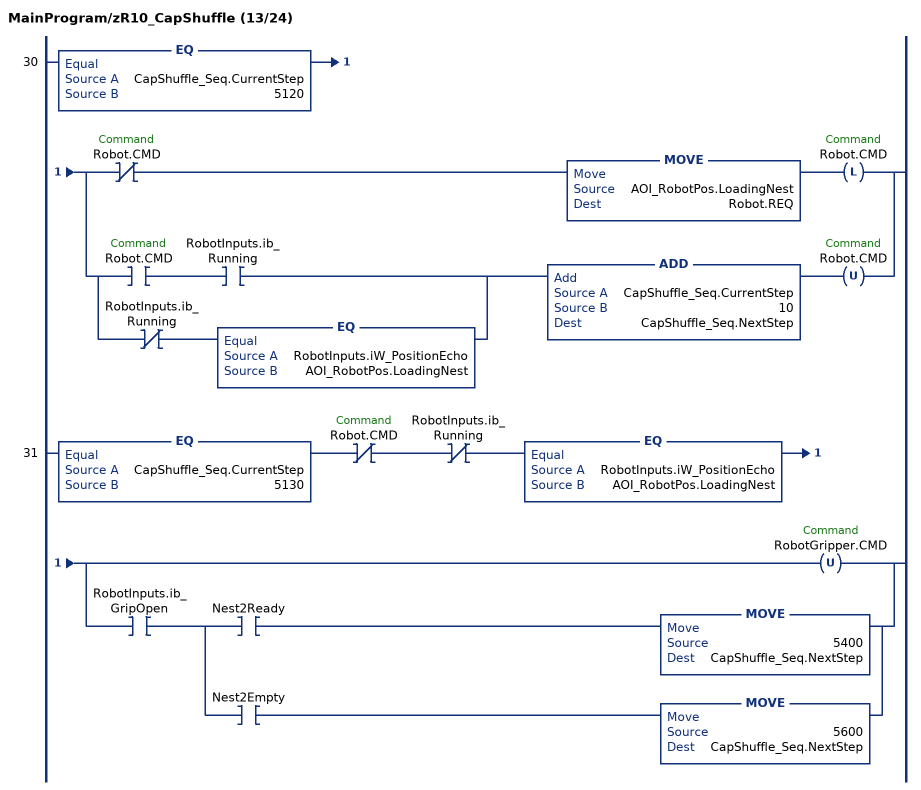
   30: EQ(CapShuffle_Seq.CurrentStep,5120)[XIO(Robot.CMD) MOVE(AOI_RobotPos.LoadingNest,Robot.REQ) OTL(Robot.CMD) ,[XIC(Robot.CMD) XIC(RobotInputs.ib_Running) ,XIO(RobotInputs.ib_Running) EQ(RobotInputs.iW_PositionEcho,AOI_RobotPos.LoadingNest) ] ADD(CapShuffle_Seq.CurrentStep,10,CapShuffle_Seq.NextStep) OTU(Robot.CMD) ];
   31: EQ(CapShuffle_Seq.CurrentStep,5130)XIO(Robot.CMD)XIO(RobotInputs.ib_Running)EQ(RobotInputs.iW_PositionEcho,AOI_RobotPos.LoadingNest)[OTU(RobotGripper.CMD) ,XIC(RobotInputs.ib_GripOpen) [XIC(Nest2Ready) MOVE(5400,CapShuffle_Seq.NextStep) ,XIC(Nest2Empty) MOVE(5600,CapShuffle_Seq.NextStep) ] ];
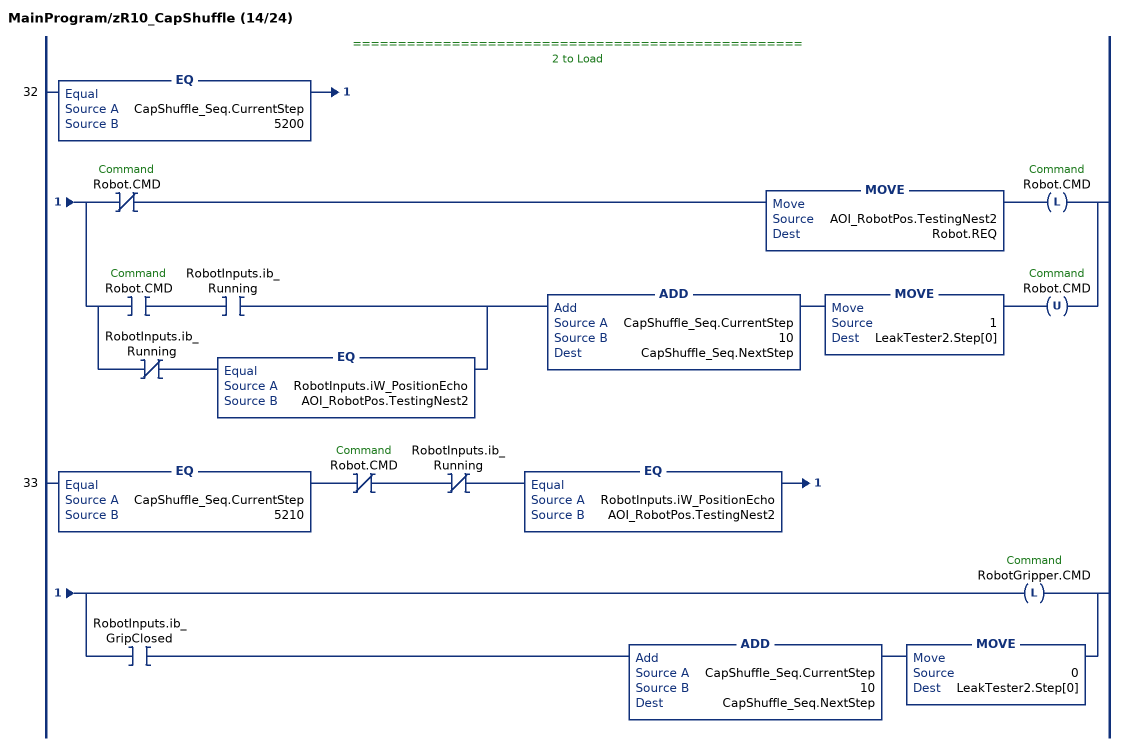
   // ==================================================
   // 2 to Load
   32: EQ(CapShuffle_Seq.CurrentStep,5200)[XIO(Robot.CMD) MOVE(AOI_RobotPos.TestingNest2,Robot.REQ) OTL(Robot.CMD) ,[XIC(Robot.CMD) XIC(RobotInputs.ib_Running) ,XIO(RobotInputs.ib_Running) EQ(RobotInputs.iW_PositionEcho,AOI_RobotPos.TestingNest2) ] ADD(CapShuffle_Seq.CurrentStep,10,CapShuffle_Seq.NextStep) MOVE(1,LeakTester2.Step[0]) OTU(Robot.CMD) ];
   33: EQ(CapShuffle_Seq.CurrentStep,5210)XIO(Robot.CMD)XIO(RobotInputs.ib_Running)EQ(RobotInputs.iW_PositionEcho,AOI_RobotPos.TestingNest2)[OTL(RobotGripper.CMD) ,XIC(RobotInputs.ib_GripClosed) ADD(CapShuffle_Seq.CurrentStep,10,CapShuffle_Seq.NextStep) MOVE(0,LeakTester2.Step[0]) ];
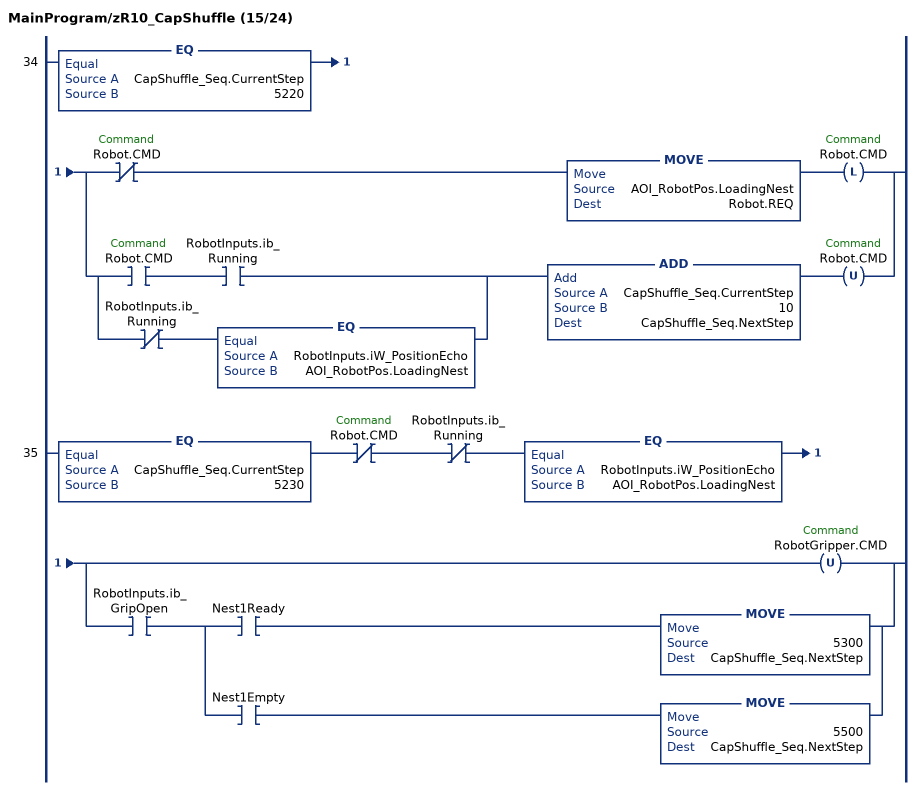
   34: EQ(CapShuffle_Seq.CurrentStep,5220)[XIO(Robot.CMD) MOVE(AOI_RobotPos.LoadingNest,Robot.REQ) OTL(Robot.CMD) ,[XIC(Robot.CMD) XIC(RobotInputs.ib_Running) ,XIO(RobotInputs.ib_Running) EQ(RobotInputs.iW_PositionEcho,AOI_RobotPos.LoadingNest) ] ADD(CapShuffle_Seq.CurrentStep,10,CapShuffle_Seq.NextStep) OTU(Robot.CMD) ];
   35: EQ(CapShuffle_Seq.CurrentStep,5230)XIO(Robot.CMD)XIO(RobotInputs.ib_Running)EQ(RobotInputs.iW_PositionEcho,AOI_RobotPos.LoadingNest)[OTU(RobotGripper.CMD) ,XIC(RobotInputs.ib_GripOpen) [XIC(Nest1Ready) MOVE(5300,CapShuffle_Seq.NextStep) ,XIC(Nest1Empty) MOVE(5500,CapShuffle_Seq.NextStep) ] ];
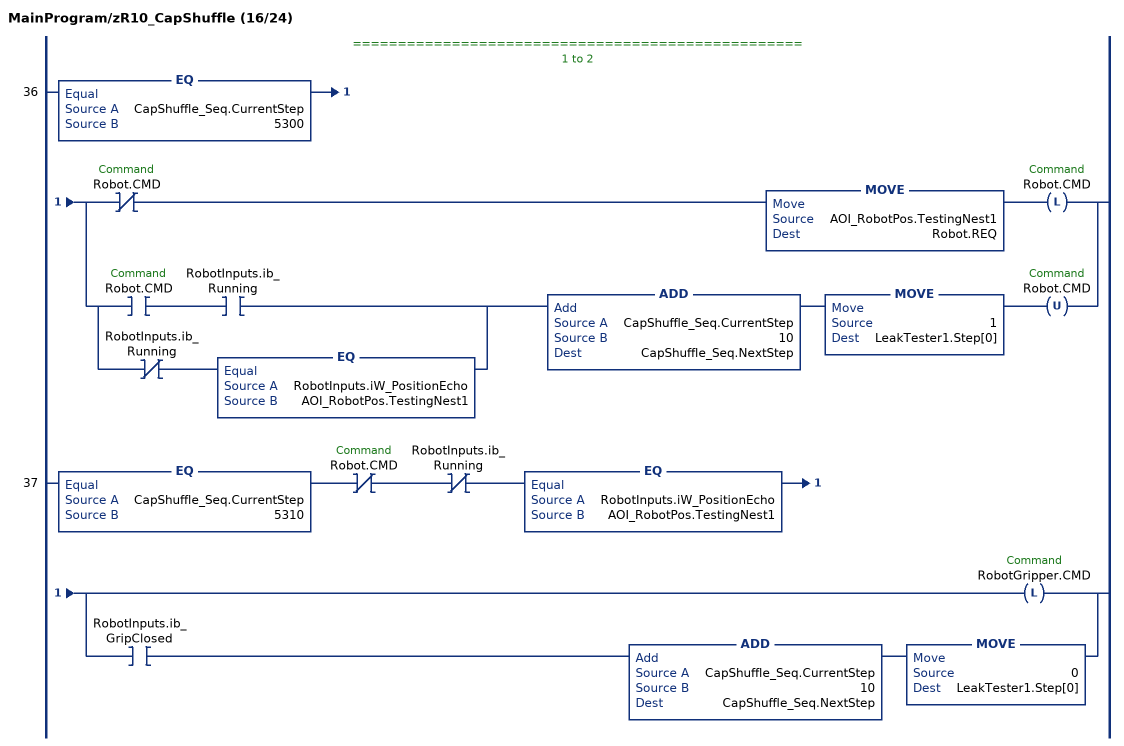
   // ==================================================
   // 1 to 2
   36: EQ(CapShuffle_Seq.CurrentStep,5300)[XIO(Robot.CMD) MOVE(AOI_RobotPos.TestingNest1,Robot.REQ) OTL(Robot.CMD) ,[XIC(Robot.CMD) XIC(RobotInputs.ib_Running) ,XIO(RobotInputs.ib_Running) EQ(RobotInputs.iW_PositionEcho,AOI_RobotPos.TestingNest1) ] ADD(CapShuffle_Seq.CurrentStep,10,CapShuffle_Seq.NextStep) MOVE(1,LeakTester1.Step[0]) OTU(Robot.CMD) ];
   37: EQ(CapShuffle_Seq.CurrentStep,5310)XIO(Robot.CMD)XIO(RobotInputs.ib_Running)EQ(RobotInputs.iW_PositionEcho,AOI_RobotPos.TestingNest1)[OTL(RobotGripper.CMD) ,XIC(RobotInputs.ib_GripClosed) ADD(CapShuffle_Seq.CurrentStep,10,CapShuffle_Seq.NextStep) MOVE(0,LeakTester1.Step[0]) ];
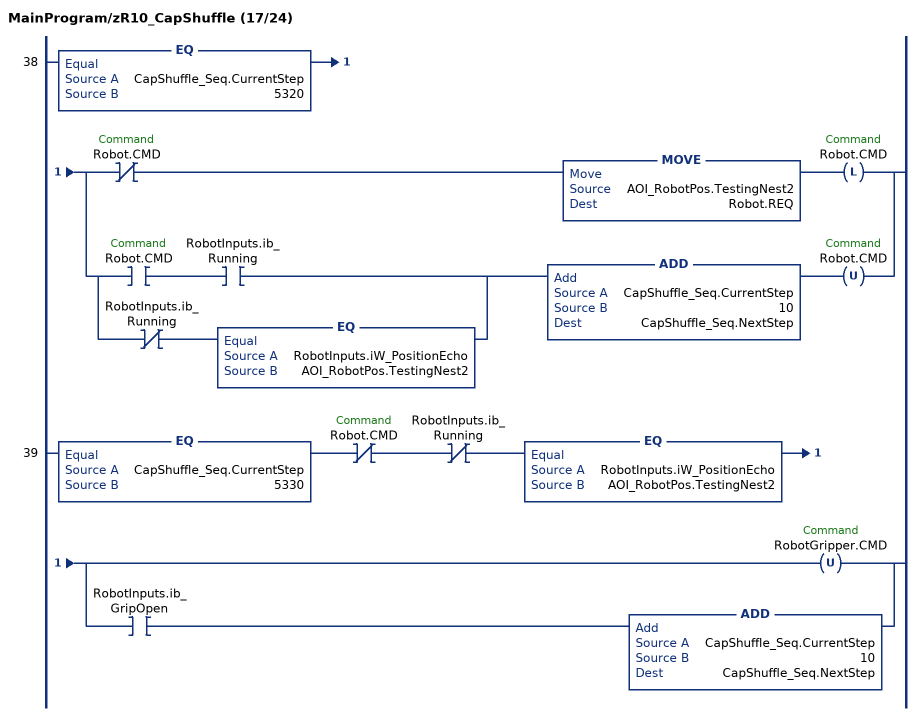
   38: EQ(CapShuffle_Seq.CurrentStep,5320)[XIO(Robot.CMD) MOVE(AOI_RobotPos.TestingNest2,Robot.REQ) OTL(Robot.CMD) ,[XIC(Robot.CMD) XIC(RobotInputs.ib_Running) ,XIO(RobotInputs.ib_Running) EQ(RobotInputs.iW_PositionEcho,AOI_RobotPos.TestingNest2) ] ADD(CapShuffle_Seq.CurrentStep,10,CapShuffle_Seq.NextStep) OTU(Robot.CMD) ];
   39: EQ(CapShuffle_Seq.CurrentStep,5330)XIO(Robot.CMD)XIO(RobotInputs.ib_Running)EQ(RobotInputs.iW_PositionEcho,AOI_RobotPos.TestingNest2)[OTU(RobotGripper.CMD) ,XIC(RobotInputs.ib_GripOpen) ADD(CapShuffle_Seq.CurrentStep,10,CapShuffle_Seq.NextStep) ];
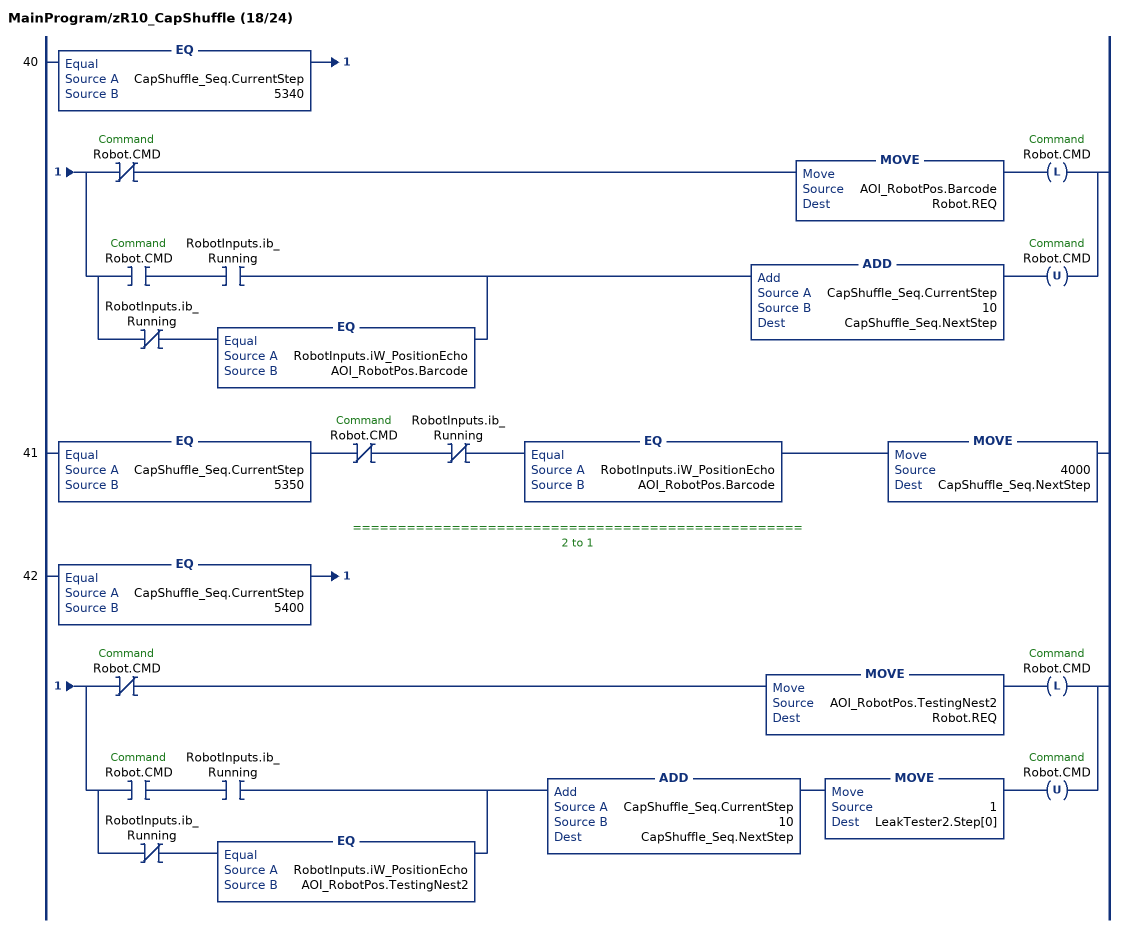
   40: EQ(CapShuffle_Seq.CurrentStep,5340)[XIO(Robot.CMD) MOVE(AOI_RobotPos.Barcode,Robot.REQ) OTL(Robot.CMD) ,[XIC(Robot.CMD) XIC(RobotInputs.ib_Running) ,XIO(RobotInputs.ib_Running) EQ(RobotInputs.iW_PositionEcho,AOI_RobotPos.Barcode) ] ADD(CapShuffle_Seq.CurrentStep,10,CapShuffle_Seq.NextStep) OTU(Robot.CMD) ];
   41: EQ(CapShuffle_Seq.CurrentStep,5350)XIO(Robot.CMD)XIO(RobotInputs.ib_Running)EQ(RobotInputs.iW_PositionEcho,AOI_RobotPos.Barcode)MOVE(4000,CapShuffle_Seq.NextStep);
   // ==================================================
   // 2 to 1
   42: EQ(CapShuffle_Seq.CurrentStep,5400)[XIO(Robot.CMD) MOVE(AOI_RobotPos.TestingNest2,Robot.REQ) OTL(Robot.CMD) ,[XIC(Robot.CMD) XIC(RobotInputs.ib_Running) ,XIO(RobotInputs.ib_Running) EQ(RobotInputs.iW_PositionEcho,AOI_RobotPos.TestingNest2) ] ADD(CapShuffle_Seq.CurrentStep,10,CapShuffle_Seq.NextStep) MOVE(1,LeakTester2.Step[0]) OTU(Robot.CMD) ];
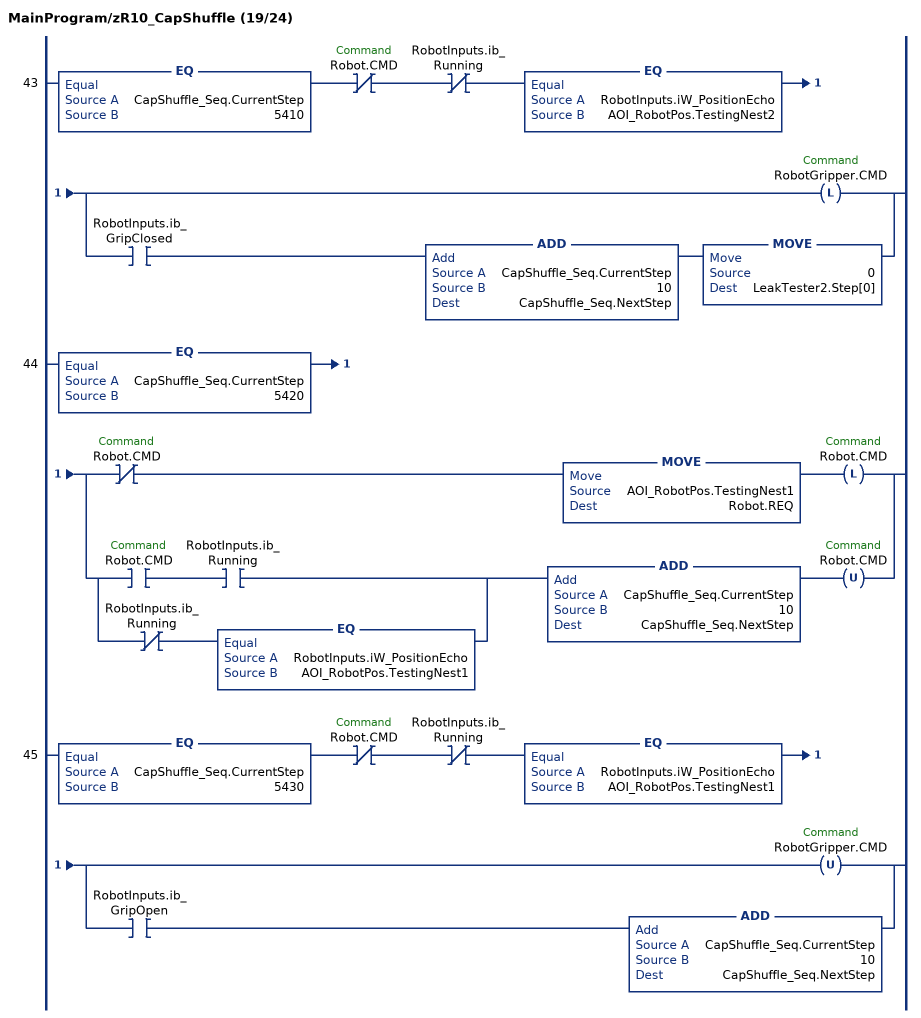
   43: EQ(CapShuffle_Seq.CurrentStep,5410)XIO(Robot.CMD)XIO(RobotInputs.ib_Running)EQ(RobotInputs.iW_PositionEcho,AOI_RobotPos.TestingNest2)[OTL(RobotGripper.CMD) ,XIC(RobotInputs.ib_GripClosed) ADD(CapShuffle_Seq.CurrentStep,10,CapShuffle_Seq.NextStep) MOVE(0,LeakTester2.Step[0]) ];
   44: EQ(CapShuffle_Seq.CurrentStep,5420)[XIO(Robot.CMD) MOVE(AOI_RobotPos.TestingNest1,Robot.REQ) OTL(Robot.CMD) ,[XIC(Robot.CMD) XIC(RobotInputs.ib_Running) ,XIO(RobotInputs.ib_Running) EQ(RobotInputs.iW_PositionEcho,AOI_RobotPos.TestingNest1) ] ADD(CapShuffle_Seq.CurrentStep,10,CapShuffle_Seq.NextStep) OTU(Robot.CMD) ];
   45: EQ(CapShuffle_Seq.CurrentStep,5430)XIO(Robot.CMD)XIO(RobotInputs.ib_Running)EQ(RobotInputs.iW_PositionEcho,AOI_RobotPos.TestingNest1)[OTU(RobotGripper.CMD) ,XIC(RobotInputs.ib_GripOpen) ADD(CapShuffle_Seq.CurrentStep,10,CapShuffle_Seq.NextStep) ];
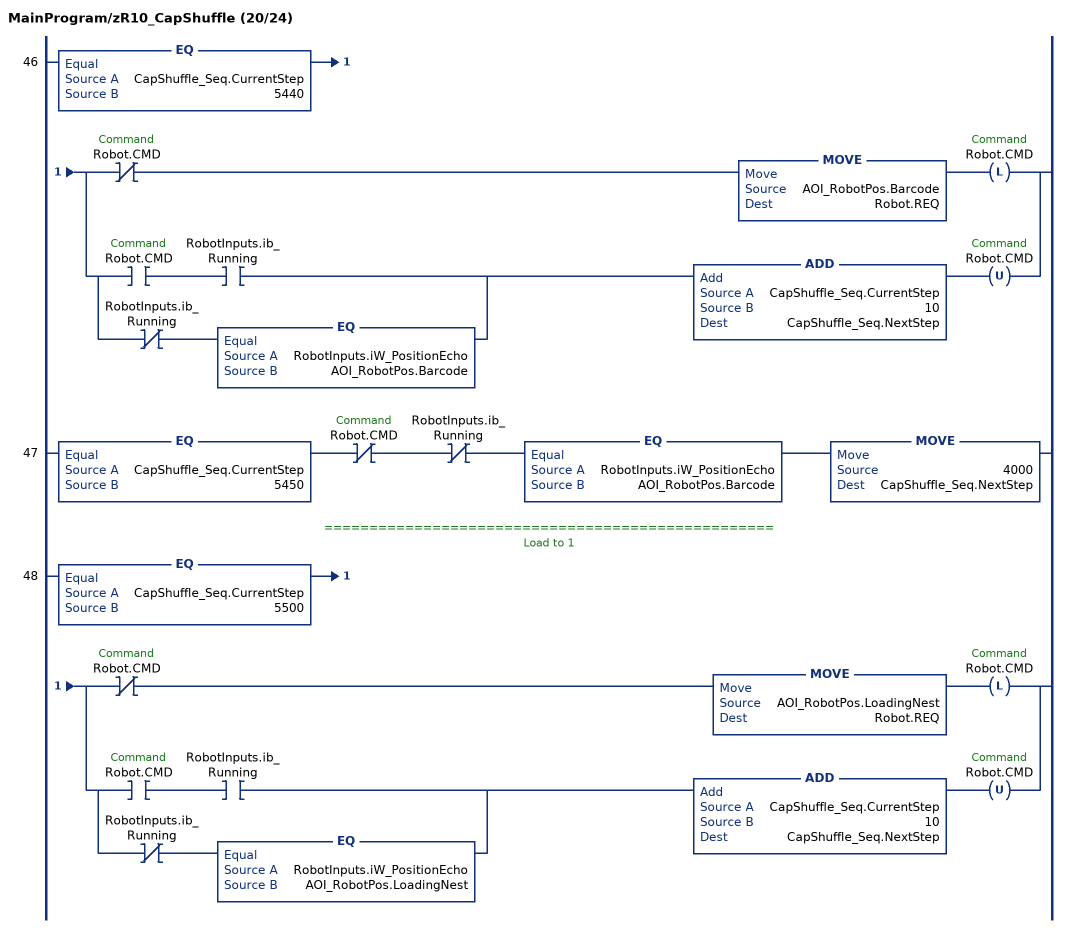
   46: EQ(CapShuffle_Seq.CurrentStep,5440)[XIO(Robot.CMD) MOVE(AOI_RobotPos.Barcode,Robot.REQ) OTL(Robot.CMD) ,[XIC(Robot.CMD) XIC(RobotInputs.ib_Running) ,XIO(RobotInputs.ib_Running) EQ(RobotInputs.iW_PositionEcho,AOI_RobotPos.Barcode) ] ADD(CapShuffle_Seq.CurrentStep,10,CapShuffle_Seq.NextStep) OTU(Robot.CMD) ];
   47: EQ(CapShuffle_Seq.CurrentStep,5450)XIO(Robot.CMD)XIO(RobotInputs.ib_Running)EQ(RobotInputs.iW_PositionEcho,AOI_RobotPos.Barcode)MOVE(4000,CapShuffle_Seq.NextStep);
   // ==================================================
   // Load to 1
   48: EQ(CapShuffle_Seq.CurrentStep,5500)[XIO(Robot.CMD) MOVE(AOI_RobotPos.LoadingNest,Robot.REQ) OTL(Robot.CMD) ,[XIC(Robot.CMD) XIC(RobotInputs.ib_Running) ,XIO(RobotInputs.ib_Running) EQ(RobotInputs.iW_PositionEcho,AOI_RobotPos.LoadingNest) ] ADD(CapShuffle_Seq.CurrentStep,10,CapShuffle_Seq.NextStep) OTU(Robot.CMD) ];
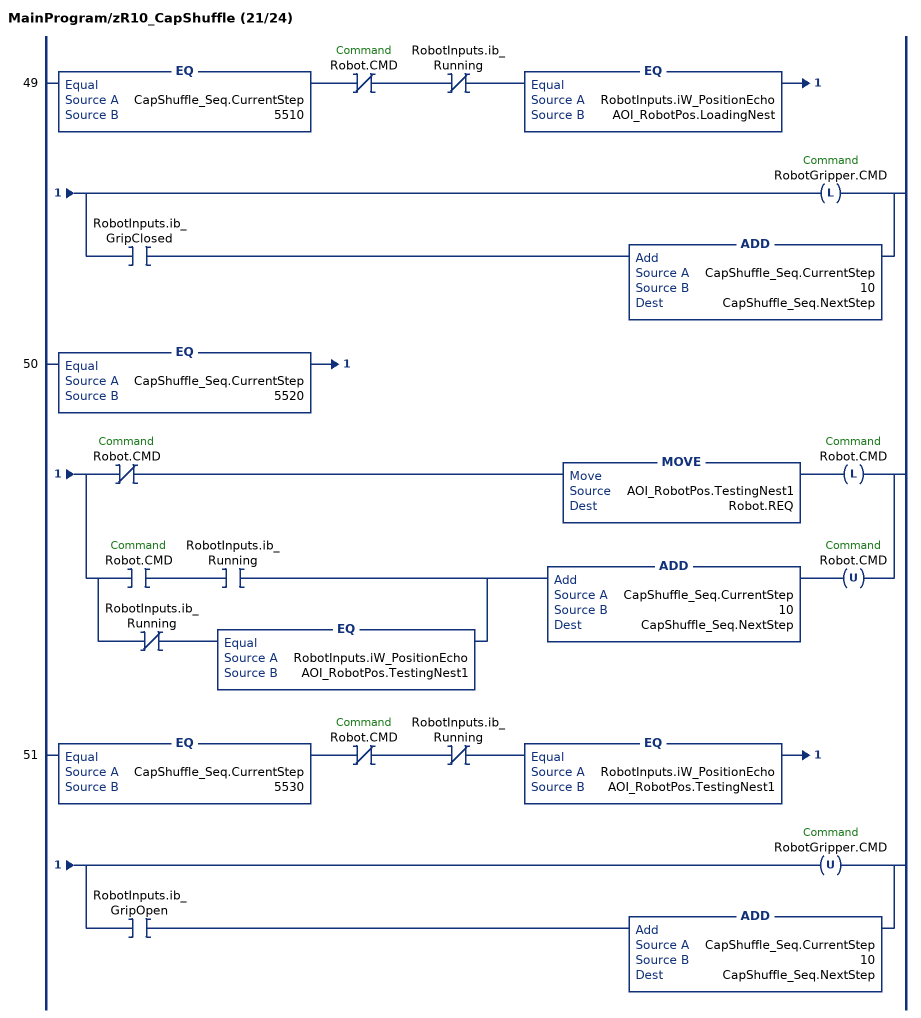
   49: EQ(CapShuffle_Seq.CurrentStep,5510)XIO(Robot.CMD)XIO(RobotInputs.ib_Running)EQ(RobotInputs.iW_PositionEcho,AOI_RobotPos.LoadingNest)[OTL(RobotGripper.CMD) ,XIC(RobotInputs.ib_GripClosed) ADD(CapShuffle_Seq.CurrentStep,10,CapShuffle_Seq.NextStep) ];
   50: EQ(CapShuffle_Seq.CurrentStep,5520)[XIO(Robot.CMD) MOVE(AOI_RobotPos.TestingNest1,Robot.REQ) OTL(Robot.CMD) ,[XIC(Robot.CMD) XIC(RobotInputs.ib_Running) ,XIO(RobotInputs.ib_Running) EQ(RobotInputs.iW_PositionEcho,AOI_RobotPos.TestingNest1) ] ADD(CapShuffle_Seq.CurrentStep,10,CapShuffle_Seq.NextStep) OTU(Robot.CMD) ];
   51: EQ(CapShuffle_Seq.CurrentStep,5530)XIO(Robot.CMD)XIO(RobotInputs.ib_Running)EQ(RobotInputs.iW_PositionEcho,AOI_RobotPos.TestingNest1)[OTU(RobotGripper.CMD) ,XIC(RobotInputs.ib_GripOpen) ADD(CapShuffle_Seq.CurrentStep,10,CapShuffle_Seq.NextStep) ];
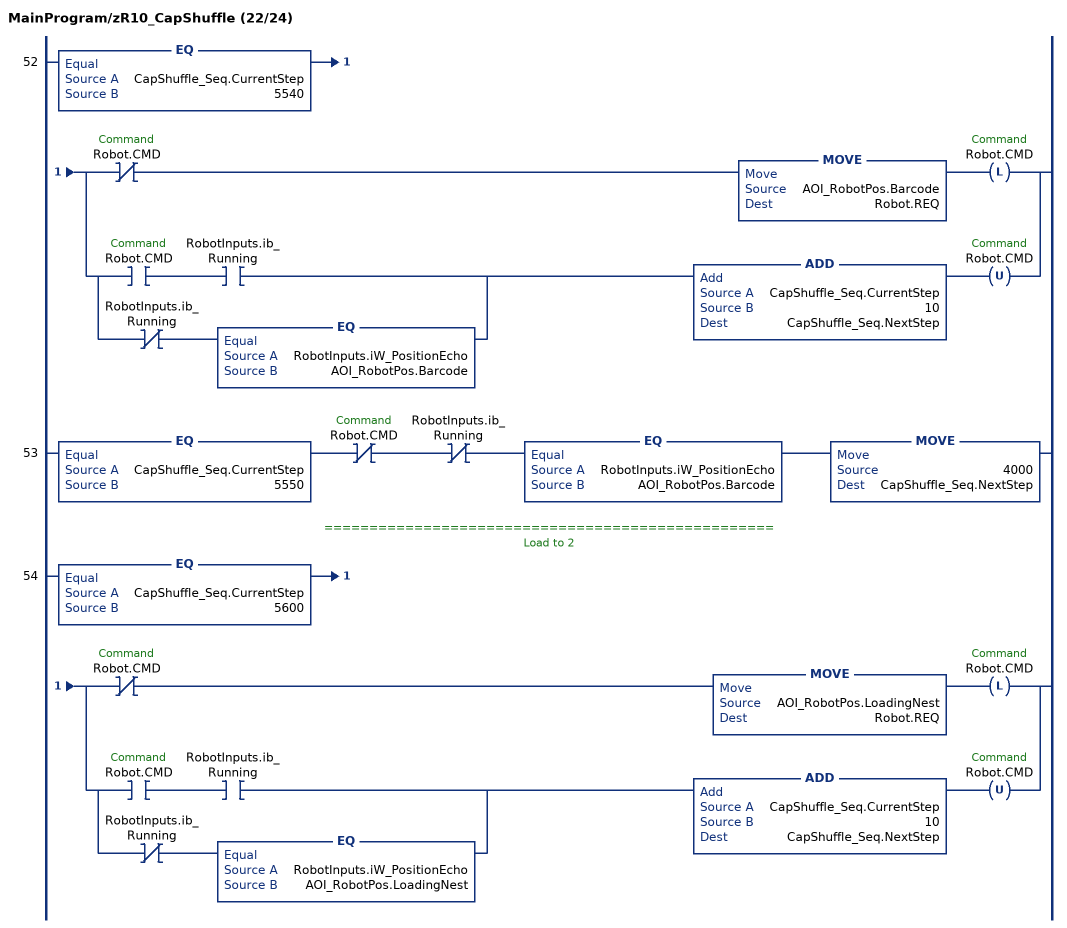
   52: EQ(CapShuffle_Seq.CurrentStep,5540)[XIO(Robot.CMD) MOVE(AOI_RobotPos.Barcode,Robot.REQ) OTL(Robot.CMD) ,[XIC(Robot.CMD) XIC(RobotInputs.ib_Running) ,XIO(RobotInputs.ib_Running) EQ(RobotInputs.iW_PositionEcho,AOI_RobotPos.Barcode) ] ADD(CapShuffle_Seq.CurrentStep,10,CapShuffle_Seq.NextStep) OTU(Robot.CMD) ];
   53: EQ(CapShuffle_Seq.CurrentStep,5550)XIO(Robot.CMD)XIO(RobotInputs.ib_Running)EQ(RobotInputs.iW_PositionEcho,AOI_RobotPos.Barcode)MOVE(4000,CapShuffle_Seq.NextStep);
   // ==================================================
   // Load to 2
   54: EQ(CapShuffle_Seq.CurrentStep,5600)[XIO(Robot.CMD) MOVE(AOI_RobotPos.LoadingNest,Robot.REQ) OTL(Robot.CMD) ,[XIC(Robot.CMD) XIC(RobotInputs.ib_Running) ,XIO(RobotInputs.ib_Running) EQ(RobotInputs.iW_PositionEcho,AOI_RobotPos.LoadingNest) ] ADD(CapShuffle_Seq.CurrentStep,10,CapShuffle_Seq.NextStep) OTU(Robot.CMD) ];
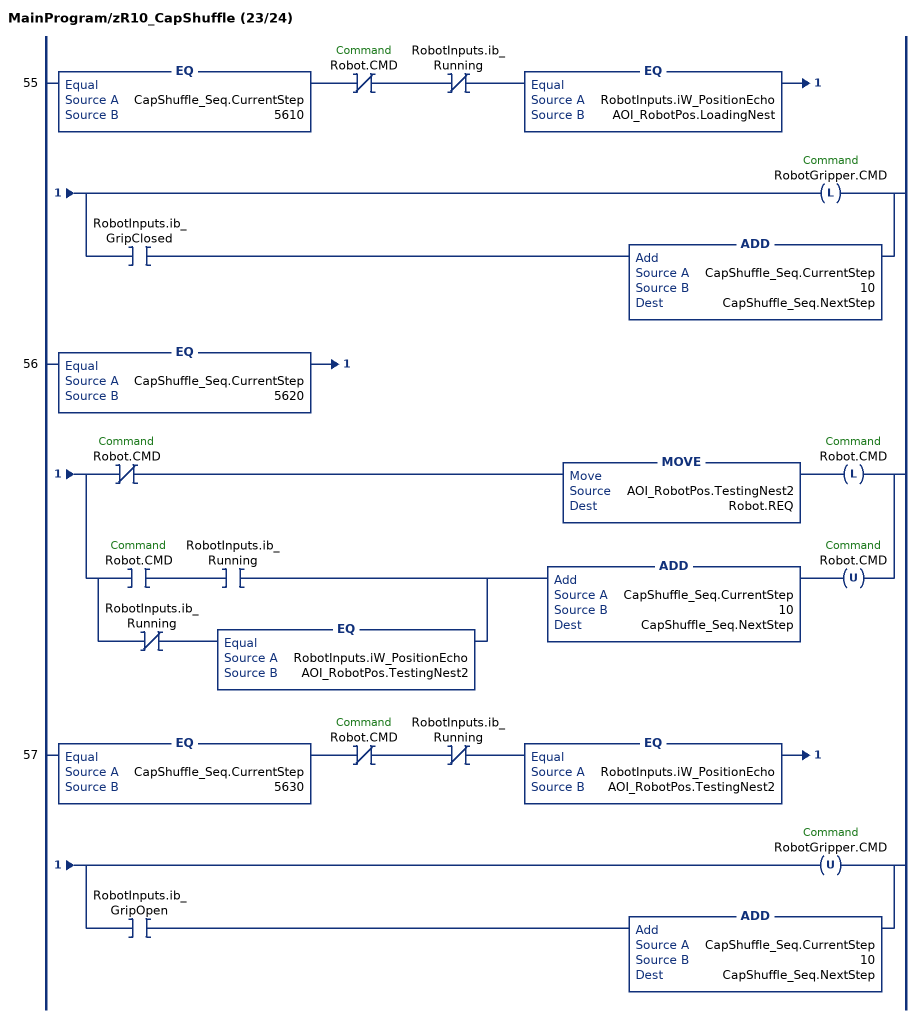
   55: EQ(CapShuffle_Seq.CurrentStep,5610)XIO(Robot.CMD)XIO(RobotInputs.ib_Running)EQ(RobotInputs.iW_PositionEcho,AOI_RobotPos.LoadingNest)[OTL(RobotGripper.CMD) ,XIC(RobotInputs.ib_GripClosed) ADD(CapShuffle_Seq.CurrentStep,10,CapShuffle_Seq.NextStep) ];
   56: EQ(CapShuffle_Seq.CurrentStep,5620)[XIO(Robot.CMD) MOVE(AOI_RobotPos.TestingNest2,Robot.REQ) OTL(Robot.CMD) ,[XIC(Robot.CMD) XIC(RobotInputs.ib_Running) ,XIO(RobotInputs.ib_Running) EQ(RobotInputs.iW_PositionEcho,AOI_RobotPos.TestingNest2) ] ADD(CapShuffle_Seq.CurrentStep,10,CapShuffle_Seq.NextStep) OTU(Robot.CMD) ];
   57: EQ(CapShuffle_Seq.CurrentStep,5630)XIO(Robot.CMD)XIO(RobotInputs.ib_Running)EQ(RobotInputs.iW_PositionEcho,AOI_RobotPos.TestingNest2)[OTU(RobotGripper.CMD) ,XIC(RobotInputs.ib_GripOpen) ADD(CapShuffle_Seq.CurrentStep,10,CapShuffle_Seq.NextStep) ];
